LIN {X 0,Y 441.877,Z 678.81,A -85,B 0,C 180,E1 7877.951,E2 7877.951} C_VEL
LIN {X 0,Y 441.94,Z 678.81,A -85,B 0,C 180,E1 7887.839,E2 7887.839} C_VEL
LIN {X 0,Y 441.992,Z 678.81,A -85,B 0,C 180,E1 7896.74,E2 7896.74} C_VEL
LIN {X 0,Y 442.419,Z 678.81,A -85,B 0,C 180,E1 7907.114,E2 7907.114} C_VEL
LIN {X 0,Y 443.093,Z 678.81,A -85,B 0,C 180,E1 7917.053,E2 7917.053} C_VEL
LIN {X 0,Y 442.904,Z 678.81,A -85,B 0,C 180,E1 7928.868,E2 7928.868} C_VEL
LIN {X 0,Y 442.435,Z 678.81,A -85,B 0,C 180,E1 7939.396,E2 7939.396} C_VEL
LIN {X 0,Y 442.136,Z 678.81,A -85,B 0,C 180,E1 7949.846,E2 7949.846} C_VEL
LIN {X 0,Y 441.88,Z 678.81,A -85,B 0,C 180,E1 7959.445,E2 7959.445} C_VEL
LIN {X 0,Y 441.823,Z 678.81,A -85,B 0,C 180,E1 7967.95,E2 7967.95} C_VEL
LIN {X 0,Y 441.903,Z 678.81,A -85,B 0,C 180,E1 7977.84,E2 7977.84} C_VEL
LIN {X 0,Y 441.903,Z 678.81,A -85,B 0,C 180,E1 7986.739,E2 7986.739} C_VEL
LIN {X 0,Y 442.388,Z 678.81,A -85,B 0,C 180,E1 7997.116,E2 7997.116} C_VEL
LIN {X 0,Y 443.106,Z 678.81,A -85,B 0,C 180,E1 8007.055,E2 8007.055} C_VEL
LIN {X 0,Y 442.18,Z 679.143,A -85,B 0,C 180,E1 8012.274,E2 8012.274} C_VEL
LIN {X 0,Y 449.727,Z 716.922,A -85,B 0,C 180,E1 8014.527,E2 8014.527} C_VEL
LIN {X 0,Y 447.081,Z 751.878,A -85,B 0,C 180,E1 8018.049,E2 8018.049} C_VEL
LIN {X 0,Y 445.187,Z 775.919,A -85,B 0,C 180,E1 8022.801,E2 8022.801} C_VEL
LIN {X 0,Y 444.517,Z 785.576,A -85,B 0,C 180,E1 8026.869,E2 8026.869} C_VEL
LIN {X 0,Y 444.32,Z 787.613,A -85,B 0,C 180,E1 8031.016,E2 8031.016} C_VEL
LIN {X 0,Y 445.139,Z 777.632,A -85,B 0,C 180,E1 8036.853,E2 8036.853} C_VEL
LIN {X 0,Y 447.345,Z 753.499,A -85,B 0,C 180,E1 8041.883,E2 8041.883} C_VEL
LIN {X 0,Y 450.088,Z 718.084,A -85,B 0,C 180,E1 8045.554,E2 8045.554} C_VEL
LIN {X 0,Y 445.324,Z 689.075,A -85,B 0,C 180,E1 8047.469,E2 8047.469} C_VEL
LIN {X 0,Y 442.183,Z 678.81,A -85,B 0,C 180,E1 8048.21,E2 8048.21} C_VEL
LIN {X 0,Y 441.838,Z 678.81,A -85,B 0,C 180,E1 8057.952,E2 8057.952} C_VEL
LIN {X 0,Y 441.944,Z 678.81,A -85,B 0,C 180,E1 8067.844,E2 8067.844} C_VEL
LIN {X 0,Y 441.985,Z 678.81,A -85,B 0,C 180,E1 8076.744,E2 8076.744} C_VEL
LIN {X 0,Y 442.41,Z 678.81,A -85,B 0,C 180,E1 8087.118,E2 8087.118} C_VEL
LIN {X 0,Y 443.095,Z 678.81,A -85,B 0,C 180,E1 8097.057,E2 8097.057} C_VEL
LIN {X 0,Y 443.049,Z 678.81,A -85,B 0,C 180,E1 8106.888,E2 8106.888} C_VEL
LIN {X 0,Y 442.491,Z 678.81,A -85,B 0,C 180,E1 8116.952,E2 8116.952} C_VEL
LIN {X 0,Y 442.197,Z 678.81,A -85,B 0,C 180,E1 8127.604,E2 8127.604} C_VEL
LIN {X 0,Y 442.091,Z 678.81,A -85,B 0,C 180,E1 8136.926,E2 8136.926} C_VEL
LIN {X 0,Y 441.903,Z 678.81,A -85,B 0,C 180,E1 8147.596,E2 8147.596} C_VEL
LIN {X 0,Y 441.983,Z 678.81,A -85,B 0,C 180,E1 8157.846,E2 8157.846} C_VEL
LIN {X 0,Y 442.499,Z 680.168,A -85,B 0,C 180,E1 8161.703,E2 8161.703} C_VEL
LIN {X 0,Y 454.771,Z 724.239,A -85,B 0,C 180,E1 8163.121,E2 8163.121} C_VEL
LIN {X 0,Y 452.774,Z 780.472,A -85,B 0,C 180,E1 8164.766,E2 8164.766} C_VEL
LIN {X 0,Y 452.64,Z 781.9,A -85,B 0,C 180,E1 8164.834,E2 8164.834} C_VEL
LIN {X 0,Y 442.739,Z 813.411,A -85,B 0,C 180,E1 8166.492,E2 8166.492} C_VEL
LIN {X 0,Y 438.607,Z 858.556,A -85,B 0,C 180,E1 8171.213,E2 8171.213} C_VEL
LIN {X 0,Y 436.435,Z 891.911,A -85,B 0,C 180,E1 8177.193,E2 8177.193} C_VEL
LIN {X 0,Y 436.07,Z 912.085,A -85,B 0,C 180,E1 8184.007,E2 8184.007} C_VEL
LIN {X 0,Y 435.871,Z 917.371,A -85,B 0,C 180,E1 8190.997,E2 8190.997} C_VEL
LIN {X 0,Y 435.685,Z 909.052,A -85,B 0,C 180,E1 8197.505,E2 8197.505} C_VEL
LIN {X 0,Y 436.677,Z 886.527,A -85,B 0,C 180,E1 8204.079,E2 8204.079} C_VEL
LIN {X 0,Y 439.545,Z 849.957,A -85,B 0,C 180,E1 8209.934,E2 8209.934} C_VEL
LIN {X 0,Y 443.584,Z 803.083,A -85,B 0,C 180,E1 8214.238,E2 8214.238} C_VEL
LIN {X 0,Y 446.827,Z 750.347,A -85,B 0,C 180,E1 8216.674,E2 8216.674} C_VEL
LIN {X 0,Y 444.835,Z 713.614,A -85,B 0,C 180,E1 8217.491,E2 8217.491} C_VEL
LIN {X 0,Y 433.969,Z 678.81,A -85,B 0,C 180,E1 8218.814,E2 8218.814} C_VEL
LIN {X 0,Y 433.799,Z 678.81,A -85,B 0,C 180,E1 8228.076,E2 8228.076} C_VEL
LIN {X 0,Y 433.797,Z 678.81,A -85,B 0,C 180,E1 8238.775,E2 8238.775} C_VEL
LIN {X 0,Y 433.951,Z 678.81,A -85,B 0,C 180,E1 8249.527,E2 8249.527} C_VEL
LIN {X 0,Y 434.098,Z 678.81,A -85,B 0,C 180,E1 8260.6,E2 8260.6} C_VEL
LIN {X 0,Y 434.846,Z 678.81,A -85,B 0,C 180,E1 8270.962,E2 8270.962} C_VEL
LIN {X 0,Y 435.297,Z 678.81,A -85,B 0,C 180,E1 8278.999,E2 8278.999} C_VEL
LIN {X 0,Y 434.769,Z 678.81,A -85,B 0,C 180,E1 8291.067,E2 8291.067} C_VEL
LIN {X 0,Y 434.349,Z 678.81,A -85,B 0,C 180,E1 8301.521,E2 8301.521} C_VEL
LIN {X 0,Y 433.969,Z 678.81,A -85,B 0,C 180,E1 8311.048,E2 8311.048} C_VEL
LIN {X 0,Y 433.777,Z 678.81,A -85,B 0,C 180,E1 8321.222,E2 8321.222} C_VEL
LIN {X 0,Y 433.68,Z 678.81,A -85,B 0,C 180,E1 8331.937,E2 8331.937} C_VEL
LIN {X 0,Y 433.976,Z 678.81,A -85,B 0,C 180,E1 8341.831,E2 8341.831} C_VEL
LIN {X 0,Y 434.276,Z 678.81,A -85,B 0,C 180,E1 8352.721,E2 8352.721} C_VEL
LIN {X 0,Y 434.938,Z 678.81,A -85,B 0,C 180,E1 8362.986,E2 8362.986} C_VEL
LIN {X 0,Y 434.25,Z 678.81,A -85,B 0,C 180,E1 8371.815,E2 8371.815} C_VEL
LIN {X 0,Y 442.066,Z 718.948,A -85,B 0,C 180,E1 8374.298,E2 8374.298} C_VEL
LIN {X 0,Y 439.279,Z 753.815,A -85,B 0,C 180,E1 8377.943,E2 8377.943} C_VEL
LIN {X 0,Y 437.249,Z 778.246,A -85,B 0,C 180,E1 8383.038,E2 8383.038} C_VEL
LIN {X 0,Y 436.541,Z 787.188,A -85,B 0,C 180,E1 8387.187,E2 8387.187} C_VEL
LIN {X 0,Y 436.779,Z 786.5,A -85,B 0,C 180,E1 8393.551,E2 8393.551} C_VEL
LIN {X 0,Y 438.438,Z 770.38,A -85,B 0,C 180,E1 8399.269,E2 8399.269} C_VEL
LIN {X 0,Y 441.15,Z 741.521,A -85,B 0,C 180,E1 8403.838,E2 8403.838} C_VEL
LIN {X 0,Y 441.511,Z 704.131,A -85,B 0,C 180,E1 8406.978,E2 8406.978} C_VEL
LIN {X 0,Y 434.104,Z 678.81,A -85,B 0,C 180,E1 8408.703,E2 8408.703} C_VEL
LIN {X 0,Y 433.703,Z 678.81,A -85,B 0,C 180,E1 8419.66,E2 8419.66} C_VEL
LIN {X 0,Y 433.978,Z 678.81,A -85,B 0,C 180,E1 8429.534,E2 8429.534} C_VEL
LIN {X 0,Y 434.092,Z 678.81,A -85,B 0,C 180,E1 8440.604,E2 8440.604} C_VEL
LIN {X 0,Y 434.849,Z 678.81,A -85,B 0,C 180,E1 8450.966,E2 8450.966} C_VEL
LIN {X 0,Y 435.015,Z 678.81,A -85,B 0,C 180,E1 8461.002,E2 8461.002} C_VEL
LIN {X 0,Y 434.693,Z 678.81,A -85,B 0,C 180,E1 8471.073,E2 8471.073} C_VEL
LIN {X 0,Y 434.356,Z 678.81,A -85,B 0,C 180,E1 8481.525,E2 8481.525} C_VEL
LIN {X 0,Y 434.026,Z 678.81,A -85,B 0,C 180,E1 8491.06,E2 8491.06} C_VEL
LIN {X 0,Y 433.912,Z 678.81,A -85,B 0,C 180,E1 8501.242,E2 8501.242} C_VEL
LIN {X 0,Y 433.872,Z 678.81,A -85,B 0,C 180,E1 8512.259,E2 8512.259} C_VEL
LIN {X 0,Y 434.464,Z 680.417,A -85,B 0,C 180,E1 8521.215,E2 8521.215} C_VEL
LIN {X 0,Y 447.42,Z 725.661,A -85,B 0,C 180,E1 8522.749,E2 8522.749} C_VEL
LIN {X 0,Y 445.189,Z 781.406,A -85,B 0,C 180,E1 8524.463,E2 8524.463} C_VEL
LIN {X 0,Y 442.739,Z 813.411,A -85,B 0,C 180,E1 8526.492,E2 8526.492} C_VEL
LIN {X 0,Y 432.436,Z 841.873,A -85,B 0,C 180,E1 8528.923,E2 8528.923} C_VEL
LIN {X 0,Y 429.299,Z 879.992,A -85,B 0,C 180,E1 8534.626,E2 8534.626} C_VEL
LIN {X 0,Y 427.929,Z 905.255,A -85,B 0,C 180,E1 8541.332,E2 8541.332} C_VEL
LIN {X 0,Y 427.867,Z 914.935,A -85,B 0,C 180,E1 8546.95,E2 8546.95} C_VEL
LIN {X 0,Y 428.123,Z 913.998,A -85,B 0,C 180,E1 8554.065,E2 8554.065} C_VEL
LIN {X 0,Y 428.103,Z 897.643,A -85,B 0,C 180,E1 8561.243,E2 8561.243} C_VEL
LIN {X 0,Y 429.981,Z 868.516,A -85,B 0,C 180,E1 8567.457,E2 8567.457} C_VEL
LIN {X 0,Y 433.947,Z 825.892,A -85,B 0,C 180,E1 8572.695,E2 8572.695} C_VEL
LIN {X 0,Y 438.014,Z 774.746,A -85,B 0,C 180,E1 8576.137,E2 8576.137} C_VEL
LIN {X 0,Y 438.357,Z 718.264,A -85,B 0,C 180,E1 8577.745,E2 8577.745} C_VEL
LIN {X 0,Y 425.957,Z 678.81,A -85,B 0,C 180,E1 8579.198,E2 8579.198} C_VEL
LIN {X 0,Y 425.769,Z 678.81,A -85,B 0,C 180,E1 8589.969,E2 8589.969} C_VEL
LIN {X 0,Y 425.735,Z 678.81,A -85,B 0,C 180,E1 8600.029,E2 8600.029} C_VEL
LIN {X 0,Y 425.916,Z 678.81,A -85,B 0,C 180,E1 8610.802,E2 8610.802} C_VEL
LIN {X 0,Y 426.102,Z 678.81,A -85,B 0,C 180,E1 8620.697,E2 8620.697} C_VEL
LIN {X 0,Y 426.796,Z 678.81,A -85,B 0,C 180,E1 8630.79,E2 8630.79} C_VEL
LIN {X 0,Y 427.307,Z 678.81,A -85,B 0,C 180,E1 8638.98,E2 8638.98} C_VEL
LIN {X 0,Y 426.731,Z 678.81,A -85,B 0,C 180,E1 8651.278,E2 8651.278} C_VEL
LIN {X 0,Y 426.325,Z 678.81,A -85,B 0,C 180,E1 8661.947,E2 8661.947} C_VEL
LIN {X 0,Y 425.888,Z 678.81,A -85,B 0,C 180,E1 8673.137,E2 8673.137} C_VEL
LIN {X 0,Y 425.745,Z 678.81,A -85,B 0,C 180,E1 8684.033,E2 8684.033} C_VEL
LIN {X 0,Y 425.692,Z 678.81,A -85,B 0,C 180,E1 8693.97,E2 8693.97} C_VEL
LIN {X 0,Y 425.958,Z 678.81,A -85,B 0,C 180,E1 8703.555,E2 8703.555} C_VEL
LIN {X 0,Y 426.356,Z 678.81,A -85,B 0,C 180,E1 8714.517,E2 8714.517} C_VEL
LIN {X 0,Y 426.839,Z 678.81,A -85,B 0,C 180,E1 8724.901,E2 8724.901} C_VEL
LIN {X 0,Y 426.588,Z 680.772,A -85,B 0,C 180,E1 8731.51,E2 8731.51} C_VEL
LIN {X 0,Y 434.61,Z 718.951,A -85,B 0,C 180,E1 8733.914,E2 8733.914} C_VEL
LIN {X 0,Y 431.635,Z 753.982,A -85,B 0,C 180,E1 8737.576,E2 8737.576} C_VEL
LIN {X 0,Y 429.438,Z 778.919,A -85,B 0,C 180,E1 8742.76,E2 8742.76} C_VEL
LIN {X 0,Y 428.589,Z 788.786,A -85,B 0,C 180,E1 8747.516,E2 8747.516} C_VEL
LIN {X 0,Y 428.848,Z 788.247,A -85,B 0,C 180,E1 8753.23,E2 8753.23} C_VEL
LIN {X 0,Y 430.38,Z 773.875,A -85,B 0,C 180,E1 8758.929,E2 8758.929} C_VEL
LIN {X 0,Y 433.163,Z 747.105,A -85,B 0,C 180,E1 8763.627,E2 8763.627} C_VEL
LIN {X 0,Y 435.057,Z 709.963,A -85,B 0,C 180,E1 8767.024,E2 8767.024} C_VEL
LIN {X 0,Y 426.081,Z 678.81,A -85,B 0,C 180,E1 8769.062,E2 8769.062} C_VEL
LIN {X 0,Y 425.673,Z 678.81,A -85,B 0,C 180,E1 8780.039,E2 8780.039} C_VEL
LIN {X 0,Y 425.971,Z 678.81,A -85,B 0,C 180,E1 8791.253,E2 8791.253} C_VEL
LIN {X 0,Y 426.21,Z 678.81,A -85,B 0,C 180,E1 8802.384,E2 8802.384} C_VEL
LIN {X 0,Y 426.906,Z 678.81,A -85,B 0,C 180,E1 8812.855,E2 8812.855} C_VEL
LIN {X 0,Y 427.024,Z 678.81,A -85,B 0,C 180,E1 8821.02,E2 8821.02} C_VEL
LIN {X 0,Y 426.672,Z 678.81,A -85,B 0,C 180,E1 8831.284,E2 8831.284} C_VEL
LIN {X 0,Y 426.324,Z 678.81,A -85,B 0,C 180,E1 8841.951,E2 8841.951} C_VEL
LIN {X 0,Y 426.006,Z 678.81,A -85,B 0,C 180,E1 8853.161,E2 8853.161} C_VEL
LIN {X 0,Y 425.864,Z 678.81,A -85,B 0,C 180,E1 8864.023,E2 8864.023} C_VEL
LIN {X 0,Y 425.827,Z 678.81,A -85,B 0,C 180,E1 8873.983,E2 8873.983} C_VEL
LIN {X 0,Y 426.385,Z 680.424,A -85,B 0,C 180,E1 8880.699,E2 8880.699} C_VEL
LIN {X 0,Y 440.084,Z 727.574,A -85,B 0,C 180,E1 8882.364,E2 8882.364} C_VEL
LIN {X 0,Y 437.615,Z 782.033,A -85,B 0,C 180,E1 8884.133,E2 8884.133} C_VEL
LIN {X 0,Y 433.379,Z 832.186,A -85,B 0,C 180,E1 8887.881,E2 8887.881} C_VEL
LIN {X 0,Y 432.436,Z 841.873,A -85,B 0,C 180,E1 8888.923,E2 8888.923} C_VEL
LIN {X 0,Y 422.308,Z 866.311,A -85,B 0,C 180,E1 8892.084,E2 8892.084} C_VEL
LIN {X 0,Y 420.41,Z 896.275,A -85,B 0,C 180,E1 8898.549,E2 8898.549} C_VEL
LIN {X 0,Y 420.05,Z 912.726,A -85,B 0,C 180,E1 8905.856,E2 8905.856} C_VEL
LIN {X 0,Y 420.028,Z 915.036,A -85,B 0,C 180,E1 8911.035,E2 8911.035} C_VEL
LIN {X 0,Y 419.87,Z 906.627,A -85,B 0,C 180,E1 8917.79,E2 8917.79} C_VEL
LIN {X 0,Y 421.133,Z 882.605,A -85,B 0,C 180,E1 8924.877,E2 8924.877} C_VEL
LIN {X 0,Y 424.28,Z 845.522,A -85,B 0,C 180,E1 8930.82,E2 8930.82} C_VEL
LIN {X 0,Y 428.604,Z 798.386,A -85,B 0,C 180,E1 8935.148,E2 8935.148} C_VEL
LIN {X 0,Y 432.027,Z 745.581,A -85,B 0,C 180,E1 8937.527,E2 8937.527} C_VEL
LIN {X 0,Y 429.827,Z 716.725,A -85,B 0,C 180,E1 8938.211,E2 8938.211} C_VEL
LIN {X 0,Y 417.896,Z 678.81,A -85,B 0,C 180,E1 8939.608,E2 8939.608} C_VEL
LIN {X 0,Y 417.75,Z 678.81,A -85,B 0,C 180,E1 8949.473,E2 8949.473} C_VEL
LIN {X 0,Y 417.709,Z 678.81,A -85,B 0,C 180,E1 8960.517,E2 8960.517} C_VEL
LIN {X 0,Y 417.92,Z 678.81,A -85,B 0,C 180,E1 8970.641,E2 8970.641} C_VEL
LIN {X 0,Y 418.163,Z 678.81,A -85,B 0,C 180,E1 8982.03,E2 8982.03} C_VEL
LIN {X 0,Y 418.885,Z 678.81,A -85,B 0,C 180,E1 8992.713,E2 8992.713} C_VEL
LIN {X 0,Y 418.382,Z 678.81,A -85,B 0,C 180,E1 9001.037,E2 9001.037} C_VEL
LIN {X 0,Y 418.714,Z 678.81,A -85,B 0,C 180,E1 9011.497,E2 9011.497} C_VEL
LIN {X 0,Y 418.276,Z 678.81,A -85,B 0,C 180,E1 9022.392,E2 9022.392} C_VEL
LIN {X 0,Y 417.879,Z 678.81,A -85,B 0,C 180,E1 9031.774,E2 9031.774} C_VEL
LIN {X 0,Y 417.759,Z 678.81,A -85,B 0,C 180,E1 9042.224,E2 9042.224} C_VEL
LIN {X 0,Y 417.634,Z 678.81,A -85,B 0,C 180,E1 9053.162,E2 9053.162} C_VEL
LIN {X 0,Y 417.879,Z 678.81,A -85,B 0,C 180,E1 9063.003,E2 9063.003} C_VEL
LIN {X 0,Y 418.297,Z 678.81,A -85,B 0,C 180,E1 9074.211,E2 9074.211} C_VEL
LIN {X 0,Y 418.87,Z 678.81,A -85,B 0,C 180,E1 9085.09,E2 9085.09} C_VEL
LIN {X 0,Y 418.64,Z 680.586,A -85,B 0,C 180,E1 9091.071,E2 9091.071} C_VEL
LIN {X 0,Y 426.982,Z 720.646,A -85,B 0,C 180,E1 9093.651,E2 9093.651} C_VEL
LIN {X 0,Y 423.848,Z 755.871,A -85,B 0,C 180,E1 9097.458,E2 9097.458} C_VEL
LIN {X 0,Y 421.626,Z 779.548,A -85,B 0,C 180,E1 9102.472,E2 9102.472} C_VEL
LIN {X 0,Y 420.642,Z 790.276,A -85,B 0,C 180,E1 9107.858,E2 9107.858} C_VEL
LIN {X 0,Y 421.163,Z 787.758,A -85,B 0,C 180,E1 9114.48,E2 9114.48} C_VEL
LIN {X 0,Y 423.17,Z 770.87,A -85,B 0,C 180,E1 9120.146,E2 9120.146} C_VEL
LIN {X 0,Y 426.466,Z 740.702,A -85,B 0,C 180,E1 9124.85,E2 9124.85} C_VEL
LIN {X 0,Y 426.787,Z 707.886,A -85,B 0,C 180,E1 9127.692,E2 9127.692} C_VEL
LIN {X 0,Y 417.978,Z 678.81,A -85,B 0,C 180,E1 9129.784,E2 9129.784} C_VEL
LIN {X 0,Y 417.648,Z 678.81,A -85,B 0,C 180,E1 9140.515,E2 9140.515} C_VEL
LIN {X 0,Y 417.94,Z 678.81,A -85,B 0,C 180,E1 9150.648,E2 9150.648} C_VEL
LIN {X 0,Y 418.157,Z 678.81,A -85,B 0,C 180,E1 9162.034,E2 9162.034} C_VEL
LIN {X 0,Y 418.883,Z 678.81,A -85,B 0,C 180,E1 9172.717,E2 9172.717} C_VEL
LIN {X 0,Y 419.018,Z 678.81,A -85,B 0,C 180,E1 9181.04,E2 9181.04} C_VEL
LIN {X 0,Y 418.673,Z 678.81,A -85,B 0,C 180,E1 9191.502,E2 9191.502} C_VEL
LIN {X 0,Y 418.25,Z 678.81,A -85,B 0,C 180,E1 9202.398,E2 9202.398} C_VEL
LIN {X 0,Y 417.956,Z 678.81,A -85,B 0,C 180,E1 9211.772,E2 9211.772} C_VEL
LIN {X 0,Y 417.866,Z 678.81,A -85,B 0,C 180,E1 9222.216,E2 9222.216} C_VEL
LIN {X 0,Y 417.827,Z 678.81,A -85,B 0,C 180,E1 9233.182,E2 9233.182} C_VEL
LIN {X 0,Y 418.227,Z 680.028,A -85,B 0,C 180,E1 9240.136,E2 9240.136} C_VEL
LIN {X 0,Y 432.824,Z 725.086,A -85,B 0,C 180,E1 9241.887,E2 9241.887} C_VEL
LIN {X 0,Y 430.313,Z 780.291,A -85,B 0,C 180,E1 9243.661,E2 9243.661} C_VEL
LIN {X 0,Y 425.889,Z 829.452,A -85,B 0,C 180,E1 9247.339,E2 9247.339} C_VEL
LIN {X 0,Y 422.308,Z 866.311,A -85,B 0,C 180,E1 9252.084,E2 9252.084} C_VEL
LIN {X 0,Y 412.639,Z 886.088,A -85,B 0,C 180,E1 9255.928,E2 9255.928} C_VEL
LIN {X 0,Y 412.034,Z 906.463,A -85,B 0,C 180,E1 9262.593,E2 9262.593} C_VEL
LIN {X 0,Y 412.474,Z 913.896,A -85,B 0,C 180,E1 9268.946,E2 9268.946} C_VEL
LIN {X 0,Y 411.927,Z 908.513,A -85,B 0,C 180,E1 9276.37,E2 9276.37} C_VEL
LIN {X 0,Y 412.395,Z 889.677,A -85,B 0,C 180,E1 9283.164,E2 9283.164} C_VEL
LIN {X 0,Y 415.027,Z 856.773,A -85,B 0,C 180,E1 9289.491,E2 9289.491} C_VEL
LIN {X 0,Y 419.621,Z 812.108,A -85,B 0,C 180,E1 9294.433,E2 9294.433} C_VEL
LIN {X 0,Y 423.803,Z 760.344,A -85,B 0,C 180,E1 9297.434,E2 9297.434} C_VEL
LIN {X 0,Y 422.852,Z 719.81,A -85,B 0,C 180,E1 9298.527,E2 9298.527} C_VEL
LIN {X 0,Y 409.873,Z 678.81,A -85,B 0,C 180,E1 9299.989,E2 9299.989} C_VEL
LIN {X 0,Y 409.683,Z 678.81,A -85,B 0,C 180,E1 9310.585,E2 9310.585} C_VEL
LIN {X 0,Y 409.657,Z 678.81,A -85,B 0,C 180,E1 9319.583,E2 9319.583} C_VEL
LIN {X 0,Y 409.898,Z 678.81,A -85,B 0,C 180,E1 9330.462,E2 9330.462} C_VEL
LIN {X 0,Y 410.087,Z 678.81,A -85,B 0,C 180,E1 9341.663,E2 9341.663} C_VEL
LIN {X 0,Y 410.856,Z 678.81,A -85,B 0,C 180,E1 9352.57,E2 9352.57} C_VEL
LIN {X 0,Y 410.387,Z 678.81,A -85,B 0,C 180,E1 9361.057,E2 9361.057} C_VEL
LIN {X 0,Y 410.68,Z 678.81,A -85,B 0,C 180,E1 9371.725,E2 9371.725} C_VEL
LIN {X 0,Y 410.214,Z 678.81,A -85,B 0,C 180,E1 9382.856,E2 9382.856} C_VEL
LIN {X 0,Y 409.699,Z 678.81,A -85,B 0,C 180,E1 9393.549,E2 9393.549} C_VEL
LIN {X 0,Y 409.614,Z 678.81,A -85,B 0,C 180,E1 9403.744,E2 9403.744} C_VEL
LIN {X 0,Y 409.647,Z 678.81,A -85,B 0,C 180,E1 9414.956,E2 9414.956} C_VEL
LIN {X 0,Y 409.871,Z 678.81,A -85,B 0,C 180,E1 9425.111,E2 9425.111} C_VEL
LIN {X 0,Y 410.281,Z 678.81,A -85,B 0,C 180,E1 9436.089,E2 9436.089} C_VEL
LIN {X 0,Y 411.052,Z 678.81,A -85,B 0,C 180,E1 9446.826,E2 9446.826} C_VEL
LIN {X 0,Y 410.8,Z 680.679,A -85,B 0,C 180,E1 9450.628,E2 9450.628} C_VEL
LIN {X 0,Y 419.439,Z 721.598,A -85,B 0,C 180,E1 9453.324,E2 9453.324} C_VEL
LIN {X 0,Y 416.055,Z 757.722,A -85,B 0,C 180,E1 9457.335,E2 9457.335} C_VEL
LIN {X 0,Y 413.722,Z 781.326,A -85,B 0,C 180,E1 9462.551,E2 9462.551} C_VEL
LIN {X 0,Y 412.702,Z 791.758,A -85,B 0,C 180,E1 9468.213,E2 9468.213} C_VEL
LIN {X 0,Y 413.373,Z 788.324,A -85,B 0,C 180,E1 9474.972,E2 9474.972} C_VEL
LIN {X 0,Y 415.696,Z 769.725,A -85,B 0,C 180,E1 9480.918,E2 9480.918} C_VEL
LIN {X 0,Y 419.251,Z 739.415,A -85,B 0,C 180,E1 9485.469,E2 9485.469} C_VEL
LIN {X 0,Y 419.264,Z 708.889,A -85,B 0,C 180,E1 9488.14,E2 9488.14} C_VEL
LIN {X 0,Y 409.899,Z 678.81,A -85,B 0,C 180,E1 9490.383,E2 9490.383} C_VEL
LIN {X 0,Y 409.607,Z 678.81,A -85,B 0,C 180,E1 9499.582,E2 9499.582} C_VEL
LIN {X 0,Y 409.928,Z 678.81,A -85,B 0,C 180,E1 9510.455,E2 9510.455} C_VEL
LIN {X 0,Y 410.08,Z 678.81,A -85,B 0,C 180,E1 9521.667,E2 9521.667} C_VEL
LIN {X 0,Y 410.855,Z 678.81,A -85,B 0,C 180,E1 9532.574,E2 9532.574} C_VEL
LIN {X 0,Y 411.028,Z 678.81,A -85,B 0,C 180,E1 9541.06,E2 9541.06} C_VEL
LIN {X 0,Y 410.659,Z 678.81,A -85,B 0,C 180,E1 9551.73,E2 9551.73} C_VEL
LIN {X 0,Y 410.186,Z 678.81,A -85,B 0,C 180,E1 9562.863,E2 9562.863} C_VEL
LIN {X 0,Y 409.857,Z 678.81,A -85,B 0,C 180,E1 9573.582,E2 9573.582} C_VEL
LIN {X 0,Y 409.724,Z 678.81,A -85,B 0,C 180,E1 9583.76,E2 9583.76} C_VEL
LIN {X 0,Y 409.762,Z 678.81,A -85,B 0,C 180,E1 9594.967,E2 9594.967} C_VEL
LIN {X 0,Y 410.166,Z 679.993,A -85,B 0,C 180,E1 9599.556,E2 9599.556} C_VEL
LIN {X 0,Y 425.551,Z 729.625,A -85,B 0,C 180,E1 9601.516,E2 9601.516} C_VEL
LIN {X 0,Y 422.517,Z 784.176,A -85,B 0,C 180,E1 9603.472,E2 9603.472} C_VEL
LIN {X 0,Y 417.781,Z 833.169,A -85,B 0,C 180,E1 9607.439,E2 9607.439} C_VEL
LIN {X 0,Y 413.943,Z 873.737,A -85,B 0,C 180,E1 9613.297,E2 9613.297} C_VEL
LIN {X 0,Y 412.639,Z 886.088,A -85,B 0,C 180,E1 9615.928,E2 9615.928} C_VEL
LIN {X 0,Y 404.245,Z 900.452,A -85,B 0,C 180,E1 9620.347,E2 9620.347} C_VEL
LIN {X 0,Y 404.134,Z 911.436,A -85,B 0,C 180,E1 9626.771,E2 9626.771} C_VEL
LIN {X 0,Y 404.199,Z 911.459,A -85,B 0,C 180,E1 9633.228,E2 9633.228} C_VEL
LIN {X 0,Y 404.31,Z 898.79,A -85,B 0,C 180,E1 9640.27,E2 9640.27} C_VEL
LIN {X 0,Y 405.941,Z 870.844,A -85,B 0,C 180,E1 9647.283,E2 9647.283} C_VEL
LIN {X 0,Y 410.172,Z 830.21,A -85,B 0,C 180,E1 9653.004,E2 9653.004} C_VEL
LIN {X 0,Y 414.832,Z 780.362,A -85,B 0,C 180,E1 9656.893,E2 9656.893} C_VEL
LIN {X 0,Y 416.687,Z 725.301,A -85,B 0,C 180,E1 9658.767,E2 9658.767} C_VEL
LIN {X 0,Y 401.757,Z 678.81,A -85,B 0,C 180,E1 9660.659,E2 9660.659} C_VEL
LIN {X 0,Y 401.59,Z 678.81,A -85,B 0,C 180,E1 9671.399,E2 9671.399} C_VEL
LIN {X 0,Y 401.559,Z 678.81,A -85,B 0,C 180,E1 9681.418,E2 9681.418} C_VEL
LIN {X 0,Y 401.914,Z 678.81,A -85,B 0,C 180,E1 9692.537,E2 9692.537} C_VEL
LIN {X 0,Y 402.243,Z 678.81,A -85,B 0,C 180,E1 9704.162,E2 9704.162} C_VEL
LIN {X 0,Y 402.811,Z 678.81,A -85,B 0,C 180,E1 9714.593,E2 9714.593} C_VEL
LIN {X 0,Y 402.082,Z 678.81,A -85,B 0,C 180,E1 9723.243,E2 9723.243} C_VEL
LIN {X 0,Y 402.638,Z 678.81,A -85,B 0,C 180,E1 9731.962,E2 9731.962} C_VEL
LIN {X 0,Y 402.187,Z 678.81,A -85,B 0,C 180,E1 9743.339,E2 9743.339} C_VEL
LIN {X 0,Y 401.715,Z 678.81,A -85,B 0,C 180,E1 9753.213,E2 9753.213} C_VEL
LIN {X 0,Y 401.548,Z 678.81,A -85,B 0,C 180,E1 9764.36,E2 9764.36} C_VEL
LIN {X 0,Y 401.597,Z 678.81,A -85,B 0,C 180,E1 9774.335,E2 9774.335} C_VEL
LIN {X 0,Y 401.801,Z 678.81,A -85,B 0,C 180,E1 9784.257,E2 9784.257} C_VEL
LIN {X 0,Y 402.245,Z 678.81,A -85,B 0,C 180,E1 9795.805,E2 9795.805} C_VEL
LIN {X 0,Y 403.055,Z 678.81,A -85,B 0,C 180,E1 9806.762,E2 9806.762} C_VEL
LIN {X 0,Y 402.835,Z 679.598,A -85,B 0,C 180,E1 9810.135,E2 9810.135} C_VEL
LIN {X 0,Y 412.006,Z 721.097,A -85,B 0,C 180,E1 9812.871,E2 9812.871} C_VEL
LIN {X 0,Y 408.434,Z 757.824,A -85,B 0,C 180,E1 9816.936,E2 9816.936} C_VEL
LIN {X 0,Y 405.919,Z 782.043,A -85,B 0,C 180,E1 9822.278,E2 9822.278} C_VEL
LIN {X 0,Y 404.783,Z 793.151,A -85,B 0,C 180,E1 9828.582,E2 9828.582} C_VEL
LIN {X 0,Y 405.57,Z 788.863,A -85,B 0,C 180,E1 9835.487,E2 9835.487} C_VEL
LIN {X 0,Y 408.128,Z 769.979,A -85,B 0,C 180,E1 9841.387,E2 9841.387} C_VEL
LIN {X 0,Y 411.972,Z 739.194,A -85,B 0,C 180,E1 9845.998,E2 9845.998} C_VEL
LIN {X 0,Y 411.687,Z 709.442,A -85,B 0,C 180,E1 9848.647,E2 9848.647} C_VEL
LIN {X 0,Y 401.821,Z 678.81,A -85,B 0,C 180,E1 9850.932,E2 9850.932} C_VEL
LIN {X 0,Y 401.501,Z 678.81,A -85,B 0,C 180,E1 9861.417,E2 9861.417} C_VEL
LIN {X 0,Y 401.922,Z 678.81,A -85,B 0,C 180,E1 9872.535,E2 9872.535} C_VEL
LIN {X 0,Y 402.241,Z 678.81,A -85,B 0,C 180,E1 9884.164,E2 9884.164} C_VEL
LIN {X 0,Y 402.812,Z 678.81,A -85,B 0,C 180,E1 9894.598,E2 9894.598} C_VEL
LIN {X 0,Y 402.885,Z 678.81,A -85,B 0,C 180,E1 9903.46,E2 9903.46} C_VEL
LIN {X 0,Y 402.541,Z 678.81,A -85,B 0,C 180,E1 9914.188,E2 9914.188} C_VEL
LIN {X 0,Y 402.045,Z 678.81,A -85,B 0,C 180,E1 9925.73,E2 9925.73} C_VEL
LIN {X 0,Y 401.867,Z 678.81,A -85,B 0,C 180,E1 9935.83,E2 9935.83} C_VEL
LIN {X 0,Y 401.635,Z 678.81,A -85,B 0,C 180,E1 9947.466,E2 9947.466} C_VEL
LIN {X 0,Y 402.087,Z 679.93,A -85,B 0,C 180,E1 9958.948,E2 9958.948} C_VEL
LIN {X 0,Y 418.318,Z 730.642,A -85,B 0,C 180,E1 9961.07,E2 9961.07} C_VEL
LIN {X 0,Y 415.075,Z 784.371,A -85,B 0,C 180,E1 9963.079,E2 9963.079} C_VEL
LIN {X 0,Y 410.064,Z 833.053,A -85,B 0,C 180,E1 9967.134,E2 9967.134} C_VEL
LIN {X 0,Y 406.053,Z 872.679,A -85,B 0,C 180,E1 9973.002,E2 9973.002} C_VEL
LIN {X 0,Y 404.261,Z 900.262,A -85,B 0,C 180,E1 9980.275,E2 9980.275} C_VEL
LIN {X 0,Y 404.245,Z 900.452,A -85,B 0,C 180,E1 9980.347,E2 9980.347} C_VEL
LIN {X 0,Y 396.315,Z 908.704,A -85,B 0,C 180,E1 9985.174,E2 9985.174} C_VEL
LIN {X 0,Y 396.284,Z 911.524,A -85,B 0,C 180,E1 9991.097,E2 9991.097} C_VEL
LIN {X 0,Y 396.117,Z 902.885,A -85,B 0,C 180,E1 9998.26,E2 9998.26} C_VEL
LIN {X 0,Y 397.622,Z 878.358,A -85,B 0,C 180,E1 10005.779,E2 10005.779} C_VEL
LIN {X 0,Y 401.185,Z 841.339,A -85,B 0,C 180,E1 10011.935,E2 10011.935} C_VEL
LIN {X 0,Y 406.117,Z 793.562,A -85,B 0,C 180,E1 10016.44,E2 10016.44} C_VEL
LIN {X 0,Y 409.771,Z 741.027,A -85,B 0,C 180,E1 10018.812,E2 10018.812} C_VEL
LIN {X 0,Y 406.222,Z 717.194,A -85,B 0,C 180,E1 10019.503,E2 10019.503} C_VEL
LIN {X 0,Y 393.732,Z 678.81,A -85,B 0,C 180,E1 10021.162,E2 10021.162} C_VEL
LIN {X 0,Y 393.584,Z 678.81,A -85,B 0,C 180,E1 10032.435,E2 10032.435} C_VEL
LIN {X 0,Y 393.515,Z 678.81,A -85,B 0,C 180,E1 10043.287,E2 10043.287} C_VEL
LIN {X 0,Y 393.861,Z 678.81,A -85,B 0,C 180,E1 10053.694,E2 10053.694} C_VEL
LIN {X 0,Y 394.249,Z 678.81,A -85,B 0,C 180,E1 10065.508,E2 10065.508} C_VEL
LIN {X 0,Y 395.03,Z 678.81,A -85,B 0,C 180,E1 10076.694,E2 10076.694} C_VEL
LIN {X 0,Y 394.728,Z 678.81,A -85,B 0,C 180,E1 10089.961,E2 10089.961} C_VEL
LIN {X 0,Y 394.222,Z 678.81,A -85,B 0,C 180,E1 10101.45,E2 10101.45} C_VEL
LIN {X 0,Y 393.755,Z 678.81,A -85,B 0,C 180,E1 10111.351,E2 10111.351} C_VEL
LIN {X 0,Y 393.549,Z 678.81,A -85,B 0,C 180,E1 10122.439,E2 10122.439} C_VEL
LIN {X 0,Y 393.464,Z 678.81,A -85,B 0,C 180,E1 10133.286,E2 10133.286} C_VEL
LIN {X 0,Y 393.804,Z 678.81,A -85,B 0,C 180,E1 10143.695,E2 10143.695} C_VEL
LIN {X 0,Y 394.234,Z 678.81,A -85,B 0,C 180,E1 10155.51,E2 10155.51} C_VEL
LIN {X 0,Y 395.053,Z 678.81,A -85,B 0,C 180,E1 10166.697,E2 10166.697} C_VEL
LIN {X 0,Y 394.973,Z 679.345,A -85,B 0,C 180,E1 10169.656,E2 10169.656} C_VEL
LIN {X 0,Y 404.392,Z 723.106,A -85,B 0,C 180,E1 10172.603,E2 10172.603} C_VEL
LIN {X 0,Y 400.658,Z 759.671,A -85,B 0,C 180,E1 10176.798,E2 10176.798} C_VEL
LIN {X 0,Y 398.099,Z 783.063,A -85,B 0,C 180,E1 10182.102,E2 10182.102} C_VEL
LIN {X 0,Y 397.132,Z 792.557,A -85,B 0,C 180,E1 10186.654,E2 10186.654} C_VEL
LIN {X 0,Y 396.917,Z 794.672,A -85,B 0,C 180,E1 10191.298,E2 10191.298} C_VEL
LIN {X 0,Y 398.34,Z 785.062,A -85,B 0,C 180,E1 10197.854,E2 10197.854} C_VEL
LIN {X 0,Y 401.691,Z 761.881,A -85,B 0,C 180,E1 10203.473,E2 10203.473} C_VEL
LIN {X 0,Y 405.902,Z 725.808,A -85,B 0,C 180,E1 10207.807,E2 10207.807} C_VEL
LIN {X 0,Y 397.775,Z 690.073,A -85,B 0,C 180,E1 10210.734,E2 10210.734} C_VEL
LIN {X 0,Y 393.727,Z 678.81,A -85,B 0,C 180,E1 10211.585,E2 10211.585} C_VEL
LIN {X 0,Y 393.435,Z 678.81,A -85,B 0,C 180,E1 10222.253,E2 10222.253} C_VEL
LIN {X 0,Y 393.864,Z 678.81,A -85,B 0,C 180,E1 10233.7,E2 10233.7} C_VEL
LIN {X 0,Y 394.24,Z 678.81,A -85,B 0,C 180,E1 10245.512,E2 10245.512} C_VEL
LIN {X 0,Y 395.029,Z 678.81,A -85,B 0,C 180,E1 10256.699,E2 10256.699} C_VEL
LIN {X 0,Y 394.887,Z 678.81,A -85,B 0,C 180,E1 10267.733,E2 10267.733} C_VEL
LIN {X 0,Y 394.257,Z 678.81,A -85,B 0,C 180,E1 10279.101,E2 10279.101} C_VEL
LIN {X 0,Y 393.841,Z 678.81,A -85,B 0,C 180,E1 10289.892,E2 10289.892} C_VEL
LIN {X 0,Y 393.666,Z 678.81,A -85,B 0,C 180,E1 10301.261,E2 10301.261} C_VEL
LIN {X 0,Y 393.591,Z 678.81,A -85,B 0,C 180,E1 10312.231,E2 10312.231} C_VEL
LIN {X 0,Y 394.015,Z 680.123,A -85,B 0,C 180,E1 10318.301,E2 10318.301} C_VEL
LIN {X 0,Y 411.147,Z 729.559,A -85,B 0,C 180,E1 10320.554,E2 10320.554} C_VEL
LIN {X 0,Y 407.793,Z 783.418,A -85,B 0,C 180,E1 10322.594,E2 10322.594} C_VEL
LIN {X 0,Y 402.484,Z 831.739,A -85,B 0,C 180,E1 10326.678,E2 10326.678} C_VEL
LIN {X 0,Y 398.137,Z 871.858,A -85,B 0,C 180,E1 10332.732,E2 10332.732} C_VEL
LIN {X 0,Y 396.344,Z 899.075,A -85,B 0,C 180,E1 10340.078,E2 10340.078} C_VEL
LIN {X 0,Y 396.315,Z 908.704,A -85,B 0,C 180,E1 10345.174,E2 10345.174} C_VEL
LIN {X 0,Y 388.416,Z 910.365,A -85,B 0,C 180,E1 10350.23,E2 10350.23} C_VEL
LIN {X 0,Y 388.102,Z 903.833,A -85,B 0,C 180,E1 10357.301,E2 10357.301} C_VEL
LIN {X 0,Y 389.017,Z 882.851,A -85,B 0,C 180,E1 10364.688,E2 10364.688} C_VEL
LIN {X 0,Y 392.59,Z 846.92,A -85,B 0,C 180,E1 10371.395,E2 10371.395} C_VEL
LIN {X 0,Y 397.694,Z 801.348,A -85,B 0,C 180,E1 10376.219,E2 10376.219} C_VEL
LIN {X 0,Y 402.013,Z 748.534,A -85,B 0,C 180,E1 10379.01,E2 10379.01} C_VEL
LIN {X 0,Y 400.012,Z 722.935,A -85,B 0,C 180,E1 10379.755,E2 10379.755} C_VEL
LIN {X 0,Y 385.691,Z 678.81,A -85,B 0,C 180,E1 10381.506,E2 10381.506} C_VEL
LIN {X 0,Y 385.536,Z 678.81,A -85,B 0,C 180,E1 10393.258,E2 10393.258} C_VEL
LIN {X 0,Y 385.48,Z 678.81,A -85,B 0,C 180,E1 10403.807,E2 10403.807} C_VEL
LIN {X 0,Y 385.767,Z 678.81,A -85,B 0,C 180,E1 10413.099,E2 10413.099} C_VEL
LIN {X 0,Y 386.196,Z 678.81,A -85,B 0,C 180,E1 10425.199,E2 10425.199} C_VEL
LIN {X 0,Y 387.027,Z 678.81,A -85,B 0,C 180,E1 10436.626,E2 10436.626} C_VEL
LIN {X 0,Y 386.705,Z 678.81,A -85,B 0,C 180,E1 10450.17,E2 10450.17} C_VEL
LIN {X 0,Y 386.27,Z 678.81,A -85,B 0,C 180,E1 10459.507,E2 10459.507} C_VEL
LIN {X 0,Y 385.83,Z 678.81,A -85,B 0,C 180,E1 10469.448,E2 10469.448} C_VEL
LIN {X 0,Y 385.492,Z 678.81,A -85,B 0,C 180,E1 10480.507,E2 10480.507} C_VEL
LIN {X 0,Y 385.455,Z 678.81,A -85,B 0,C 180,E1 10490.15,E2 10490.15} C_VEL
LIN {X 0,Y 385.671,Z 678.81,A -85,B 0,C 180,E1 10500.538,E2 10500.538} C_VEL
LIN {X 0,Y 385.89,Z 678.81,A -85,B 0,C 180,E1 10510.472,E2 10510.472} C_VEL
LIN {X 0,Y 386.763,Z 678.81,A -85,B 0,C 180,E1 10522.107,E2 10522.107} C_VEL
LIN {X 0,Y 387.358,Z 680.536,A -85,B 0,C 180,E1 10529.215,E2 10529.215} C_VEL
LIN {X 0,Y 396.839,Z 724.356,A -85,B 0,C 180,E1 10532.272,E2 10532.272} C_VEL
LIN {X 0,Y 393.044,Z 759.704,A -85,B 0,C 180,E1 10536.373,E2 10536.373} C_VEL
LIN {X 0,Y 390.305,Z 783.618,A -85,B 0,C 180,E1 10541.778,E2 10541.778} C_VEL
LIN {X 0,Y 389.141,Z 794.334,A -85,B 0,C 180,E1 10547.167,E2 10547.167} C_VEL
LIN {X 0,Y 389.543,Z 793.735,A -85,B 0,C 180,E1 10554.145,E2 10554.145} C_VEL
LIN {X 0,Y 392.075,Z 778.33,A -85,B 0,C 180,E1 10560.546,E2 10560.546} C_VEL
LIN {X 0,Y 396.119,Z 750.075,A -85,B 0,C 180,E1 10565.776,E2 10565.776} C_VEL
LIN {X 0,Y 397.483,Z 714.992,A -85,B 0,C 180,E1 10569.337,E2 10569.337} C_VEL
LIN {X 0,Y 385.661,Z 678.81,A -85,B 0,C 180,E1 10572.208,E2 10572.208} C_VEL
LIN {X 0,Y 385.436,Z 678.81,A -85,B 0,C 180,E1 10583.817,E2 10583.817} C_VEL
LIN {X 0,Y 385.773,Z 678.81,A -85,B 0,C 180,E1 10593.104,E2 10593.104} C_VEL
LIN {X 0,Y 386.187,Z 678.81,A -85,B 0,C 180,E1 10605.203,E2 10605.203} C_VEL
LIN {X 0,Y 387.027,Z 678.81,A -85,B 0,C 180,E1 10616.63,E2 10616.63} C_VEL
LIN {X 0,Y 386.848,Z 678.81,A -85,B 0,C 180,E1 10627.894,E2 10627.894} C_VEL
LIN {X 0,Y 386.229,Z 678.81,A -85,B 0,C 180,E1 10639.514,E2 10639.514} C_VEL
LIN {X 0,Y 385.876,Z 678.81,A -85,B 0,C 180,E1 10649.45,E2 10649.45} C_VEL
LIN {X 0,Y 385.658,Z 678.81,A -85,B 0,C 180,E1 10660.492,E2 10660.492} C_VEL
LIN {X 0,Y 385.584,Z 678.81,A -85,B 0,C 180,E1 10670.134,E2 10670.134} C_VEL
LIN {X 0,Y 386,Z 680.419,A -85,B 0,C 180,E1 10677.627,E2 10677.627} C_VEL
LIN {X 0,Y 403.971,Z 730.228,A -85,B 0,C 180,E1 10680.057,E2 10680.057} C_VEL
LIN {X 0,Y 400.343,Z 784.423,A -85,B 0,C 180,E1 10682.209,E2 10682.209} C_VEL
LIN {X 0,Y 394.613,Z 833.198,A -85,B 0,C 180,E1 10686.525,E2 10686.525} C_VEL
LIN {X 0,Y 390.158,Z 872.152,A -85,B 0,C 180,E1 10692.679,E2 10692.679} C_VEL
LIN {X 0,Y 388.392,Z 897.915,A -85,B 0,C 180,E1 10699.873,E2 10699.873} C_VEL
LIN {X 0,Y 388.311,Z 909.112,A -85,B 0,C 180,E1 10706.639,E2 10706.639} C_VEL
LIN {X 0,Y 388.416,Z 910.365,A -85,B 0,C 180,E1 10710.23,E2 10710.23} C_VEL
LIN {X 0,Y 380.357,Z 905.814,A -85,B 0,C 180,E1 10715.363,E2 10715.363} C_VEL
LIN {X 0,Y 380.406,Z 889.626,A -85,B 0,C 180,E1 10722.674,E2 10722.674} C_VEL
LIN {X 0,Y 383.037,Z 859.02,A -85,B 0,C 180,E1 10729.679,E2 10729.679} C_VEL
LIN {X 0,Y 388.211,Z 817.137,A -85,B 0,C 180,E1 10735.158,E2 10735.158} C_VEL
LIN {X 0,Y 393.323,Z 767.327,A -85,B 0,C 180,E1 10738.677,E2 10738.677} C_VEL
LIN {X 0,Y 393.092,Z 726.098,A -85,B 0,C 180,E1 10740.107,E2 10740.107} C_VEL
LIN {X 0,Y 377.635,Z 678.81,A -85,B 0,C 180,E1 10742.203,E2 10742.203} C_VEL
LIN {X 0,Y 377.425,Z 678.81,A -85,B 0,C 180,E1 10751.933,E2 10751.933} C_VEL
LIN {X 0,Y 377.445,Z 678.81,A -85,B 0,C 180,E1 10761.629,E2 10761.629} C_VEL
LIN {X 0,Y 377.741,Z 678.81,A -85,B 0,C 180,E1 10772.479,E2 10772.479} C_VEL
LIN {X 0,Y 378.008,Z 678.81,A -85,B 0,C 180,E1 10782.473,E2 10782.473} C_VEL
LIN {X 0,Y 378.766,Z 678.81,A -85,B 0,C 180,E1 10794.249,E2 10794.249} C_VEL
LIN {X 0,Y 378.408,Z 678.81,A -85,B 0,C 180,E1 10801.147,E2 10801.147} C_VEL
LIN {X 0,Y 378.545,Z 678.81,A -85,B 0,C 180,E1 10812.736,E2 10812.736} C_VEL
LIN {X 0,Y 378.122,Z 678.81,A -85,B 0,C 180,E1 10822.411,E2 10822.411} C_VEL
LIN {X 0,Y 377.564,Z 678.81,A -85,B 0,C 180,E1 10832.861,E2 10832.861} C_VEL
LIN {X 0,Y 377.375,Z 678.81,A -85,B 0,C 180,E1 10844.727,E2 10844.727} C_VEL
LIN {X 0,Y 377.459,Z 678.81,A -85,B 0,C 180,E1 10855.507,E2 10855.507} C_VEL
LIN {X 0,Y 377.663,Z 678.81,A -85,B 0,C 180,E1 10865.044,E2 10865.044} C_VEL
LIN {X 0,Y 378.162,Z 678.81,A -85,B 0,C 180,E1 10874.88,E2 10874.88} C_VEL
LIN {X 0,Y 379.023,Z 678.81,A -85,B 0,C 180,E1 10886.557,E2 10886.557} C_VEL
LIN {X 0,Y 379.523,Z 680.686,A -85,B 0,C 180,E1 10888.714,E2 10888.714} C_VEL
LIN {X 0,Y 389.38,Z 724.121,A -85,B 0,C 180,E1 10891.804,E2 10891.804} C_VEL
LIN {X 0,Y 385.48,Z 759.71,A -85,B 0,C 180,E1 10895.932,E2 10895.932} C_VEL
LIN {X 0,Y 382.501,Z 784.167,A -85,B 0,C 180,E1 10901.442,E2 10901.442} C_VEL
LIN {X 0,Y 381.209,Z 795.729,A -85,B 0,C 180,E1 10907.372,E2 10907.372} C_VEL
LIN {X 0,Y 381.458,Z 796.101,A -85,B 0,C 180,E1 10913.127,E2 10913.127} C_VEL
LIN {X 0,Y 383.756,Z 782.968,A -85,B 0,C 180,E1 10919.843,E2 10919.843} C_VEL
LIN {X 0,Y 387.727,Z 757.822,A -85,B 0,C 180,E1 10925.241,E2 10925.241} C_VEL
LIN {X 0,Y 390.906,Z 720.318,A -85,B 0,C 180,E1 10929.46,E2 10929.46} C_VEL
LIN {X 0,Y 377.57,Z 678.81,A -85,B 0,C 180,E1 10933.158,E2 10933.158} C_VEL
LIN {X 0,Y 377.462,Z 678.81,A -85,B 0,C 180,E1 10945.506,E2 10945.506} C_VEL
LIN {X 0,Y 377.741,Z 678.81,A -85,B 0,C 180,E1 10955.051,E2 10955.051} C_VEL
LIN {X 0,Y 378.167,Z 678.81,A -85,B 0,C 180,E1 10964.882,E2 10964.882} C_VEL
LIN {X 0,Y 379.006,Z 678.81,A -85,B 0,C 180,E1 10976.559,E2 10976.559} C_VEL
LIN {X 0,Y 378.811,Z 678.81,A -85,B 0,C 180,E1 10988.063,E2 10988.063} C_VEL
LIN {X 0,Y 378.158,Z 678.81,A -85,B 0,C 180,E1 10999.948,E2 10999.948} C_VEL
LIN {X 0,Y 377.759,Z 678.81,A -85,B 0,C 180,E1 11010.265,E2 11010.265} C_VEL
LIN {X 0,Y 377.531,Z 678.81,A -85,B 0,C 180,E1 11021.958,E2 11021.958} C_VEL
LIN {X 0,Y 377.539,Z 678.81,A -85,B 0,C 180,E1 11031.619,E2 11031.619} C_VEL
LIN {X 0,Y 377.957,Z 680.545,A -85,B 0,C 180,E1 11036.912,E2 11036.912} C_VEL
LIN {X 0,Y 396.871,Z 732.705,A -85,B 0,C 180,E1 11039.585,E2 11039.585} C_VEL
LIN {X 0,Y 392.825,Z 785.873,A -85,B 0,C 180,E1 11041.834,E2 11041.834} C_VEL
LIN {X 0,Y 386.843,Z 833.945,A -85,B 0,C 180,E1 11046.274,E2 11046.274} C_VEL
LIN {X 0,Y 382.155,Z 872.659,A -85,B 0,C 180,E1 11052.673,E2 11052.673} C_VEL
LIN {X 0,Y 380.387,Z 898.188,A -85,B 0,C 180,E1 11060.238,E2 11060.238} C_VEL
LIN {X 0,Y 380.381,Z 907.958,A -85,B 0,C 180,E1 11066.569,E2 11066.569} C_VEL
LIN {X 0,Y 380.469,Z 907.879,A -85,B 0,C 180,E1 11073.43,E2 11073.43} C_VEL
LIN {X 0,Y 380.357,Z 905.814,A -85,B 0,C 180,E1 11075.363,E2 11075.363} C_VEL
LIN {X 0,Y 372.407,Z 895.39,A -85,B 0,C 180,E1 11080.407,E2 11080.407} C_VEL
LIN {X 0,Y 374.167,Z 868.339,A -85,B 0,C 180,E1 11088.014,E2 11088.014} C_VEL
LIN {X 0,Y 379.1,Z 828.531,A -85,B 0,C 180,E1 11094.224,E2 11094.224} C_VEL
LIN {X 0,Y 384.686,Z 779.848,A -85,B 0,C 180,E1 11098.415,E2 11098.415} C_VEL
LIN {X 0,Y 386.047,Z 728.911,A -85,B 0,C 180,E1 11100.48,E2 11100.48} C_VEL
LIN {X 0,Y 369.576,Z 678.81,A -85,B 0,C 180,E1 11102.663,E2 11102.663} C_VEL
LIN {X 0,Y 369.338,Z 678.81,A -85,B 0,C 180,E1 11114.018,E2 11114.018} C_VEL
LIN {X 0,Y 369.371,Z 678.81,A -85,B 0,C 180,E1 11123.43,E2 11123.43} C_VEL
LIN {X 0,Y 369.711,Z 678.81,A -85,B 0,C 180,E1 11134.465,E2 11134.465} C_VEL
LIN {X 0,Y 370.121,Z 678.81,A -85,B 0,C 180,E1 11144.54,E2 11144.54} C_VEL
LIN {X 0,Y 371.001,Z 678.81,A -85,B 0,C 180,E1 11156.48,E2 11156.48} C_VEL
LIN {X 0,Y 370.561,Z 678.81,A -85,B 0,C 180,E1 11168.239,E2 11168.239} C_VEL
LIN {X 0,Y 370.282,Z 678.81,A -85,B 0,C 180,E1 11177.9,E2 11177.9} C_VEL
LIN {X 0,Y 369.787,Z 678.81,A -85,B 0,C 180,E1 11188.159,E2 11188.159} C_VEL
LIN {X 0,Y 369.299,Z 678.81,A -85,B 0,C 180,E1 11199.563,E2 11199.563} C_VEL
LIN {X 0,Y 369.269,Z 678.81,A -85,B 0,C 180,E1 11210.433,E2 11210.433} C_VEL
LIN {X 0,Y 369.613,Z 678.81,A -85,B 0,C 180,E1 11221.976,E2 11221.976} C_VEL
LIN {X 0,Y 369.944,Z 678.81,A -85,B 0,C 180,E1 11232.082,E2 11232.082} C_VEL
LIN {X 0,Y 370.689,Z 678.81,A -85,B 0,C 180,E1 11241.762,E2 11241.762} C_VEL
LIN {X 0,Y 371.46,Z 680.825,A -85,B 0,C 180,E1 11248.185,E2 11248.185} C_VEL
LIN {X 0,Y 381.442,Z 723.815,A -85,B 0,C 180,E1 11251.279,E2 11251.279} C_VEL
LIN {X 0,Y 377.963,Z 759.698,A -85,B 0,C 180,E1 11255.472,E2 11255.472} C_VEL
LIN {X 0,Y 374.75,Z 784.698,A -85,B 0,C 180,E1 11261.09,E2 11261.09} C_VEL
LIN {X 0,Y 373.245,Z 797.214,A -85,B 0,C 180,E1 11267.754,E2 11267.754} C_VEL
LIN {X 0,Y 374.016,Z 795.139,A -85,B 0,C 180,E1 11275.216,E2 11275.216} C_VEL
LIN {X 0,Y 377.099,Z 778.318,A -85,B 0,C 180,E1 11281.795,E2 11281.795} C_VEL
LIN {X 0,Y 381.907,Z 749.064,A -85,B 0,C 180,E1 11287.065,E2 11287.065} C_VEL
LIN {X 0,Y 383.111,Z 719.259,A -85,B 0,C 180,E1 11290.218,E2 11290.218} C_VEL
LIN {X 0,Y 369.481,Z 678.81,A -85,B 0,C 180,E1 11294.047,E2 11294.047} C_VEL
LIN {X 0,Y 369.467,Z 678.81,A -85,B 0,C 180,E1 11306.325,E2 11306.325} C_VEL
LIN {X 0,Y 369.766,Z 678.81,A -85,B 0,C 180,E1 11317.431,E2 11317.431} C_VEL
LIN {X 0,Y 370.5,Z 678.81,A -85,B 0,C 180,E1 11329.381,E2 11329.381} C_VEL
LIN {X 0,Y 371.452,Z 678.81,A -85,B 0,C 180,E1 11338.832,E2 11338.832} C_VEL
LIN {X 0,Y 370.61,Z 678.81,A -85,B 0,C 180,E1 11350.621,E2 11350.621} C_VEL
LIN {X 0,Y 370.064,Z 678.81,A -85,B 0,C 180,E1 11362.68,E2 11362.68} C_VEL
LIN {X 0,Y 369.643,Z 678.81,A -85,B 0,C 180,E1 11373.663,E2 11373.663} C_VEL
LIN {X 0,Y 369.422,Z 678.81,A -85,B 0,C 180,E1 11384.038,E2 11384.038} C_VEL
LIN {X 0,Y 369.879,Z 680.499,A -85,B 0,C 180,E1 11396.134,E2 11396.134} C_VEL
LIN {X 0,Y 389.695,Z 732.585,A -85,B 0,C 180,E1 11399.013,E2 11399.013} C_VEL
LIN {X 0,Y 385.573,Z 785.64,A -85,B 0,C 180,E1 11401.336,E2 11401.336} C_VEL
LIN {X 0,Y 379.307,Z 832.881,A -85,B 0,C 180,E1 11405.79,E2 11405.79} C_VEL
LIN {X 0,Y 374.258,Z 871.789,A -85,B 0,C 180,E1 11412.359,E2 11412.359} C_VEL
LIN {X 0,Y 372.435,Z 897.031,A -85,B 0,C 180,E1 11420.028,E2 11420.028} C_VEL
LIN {X 0,Y 372.484,Z 906.906,A -85,B 0,C 180,E1 11426.616,E2 11426.616} C_VEL
LIN {X 0,Y 372.554,Z 906.63,A -85,B 0,C 180,E1 11433.562,E2 11433.562} C_VEL
LIN {X 0,Y 372.407,Z 895.39,A -85,B 0,C 180,E1 11440.407,E2 11440.407} C_VEL
LIN {X 0,Y 365.331,Z 880.019,A -85,B 0,C 180,E1 11445.253,E2 11445.253} C_VEL
LIN {X 0,Y 369.23,Z 845.167,A -85,B 0,C 180,E1 11452.239,E2 11452.239} C_VEL
LIN {X 0,Y 374.885,Z 800.282,A -85,B 0,C 180,E1 11457.34,E2 11457.34} C_VEL
LIN {X 0,Y 379.711,Z 748.395,A -85,B 0,C 180,E1 11460.302,E2 11460.302} C_VEL
LIN {X 0,Y 376.905,Z 724.668,A -85,B 0,C 180,E1 11461.148,E2 11461.148} C_VEL
LIN {X 0,Y 361.542,Z 678.81,A -85,B 0,C 180,E1 11463.227,E2 11463.227} C_VEL
LIN {X 0,Y 361.332,Z 678.81,A -85,B 0,C 180,E1 11473.866,E2 11473.866} C_VEL
LIN {X 0,Y 361.359,Z 678.81,A -85,B 0,C 180,E1 11485.458,E2 11485.458} C_VEL
LIN {X 0,Y 361.659,Z 678.81,A -85,B 0,C 180,E1 11496.504,E2 11496.504} C_VEL
LIN {X 0,Y 362.197,Z 678.81,A -85,B 0,C 180,E1 11506.674,E2 11506.674} C_VEL
LIN {X 0,Y 363.274,Z 678.81,A -85,B 0,C 180,E1 11518.801,E2 11518.801} C_VEL
LIN {X 0,Y 362.627,Z 678.81,A -85,B 0,C 180,E1 11530.853,E2 11530.853} C_VEL
LIN {X 0,Y 362.092,Z 678.81,A -85,B 0,C 180,E1 11540.868,E2 11540.868} C_VEL
LIN {X 0,Y 361.543,Z 678.81,A -85,B 0,C 180,E1 11551.646,E2 11551.646} C_VEL
LIN {X 0,Y 361.294,Z 678.81,A -85,B 0,C 180,E1 11563.872,E2 11563.872} C_VEL
LIN {X 0,Y 361.319,Z 678.81,A -85,B 0,C 180,E1 11575.459,E2 11575.459} C_VEL
LIN {X 0,Y 361.605,Z 678.81,A -85,B 0,C 180,E1 11586.504,E2 11586.504} C_VEL
LIN {X 0,Y 362.175,Z 678.81,A -85,B 0,C 180,E1 11596.676,E2 11596.676} C_VEL
LIN {X 0,Y 363.282,Z 680.345,A -85,B 0,C 180,E1 11607.606,E2 11607.606} C_VEL
LIN {X 0,Y 373.739,Z 724.862,A -85,B 0,C 180,E1 11610.878,E2 11610.878} C_VEL
LIN {X 0,Y 370.185,Z 761.47,A -85,B 0,C 180,E1 11615.292,E2 11615.292} C_VEL
LIN {X 0,Y 366.738,Z 787.036,A -85,B 0,C 180,E1 11621.336,E2 11621.336} C_VEL
LIN {X 0,Y 365.301,Z 798.693,A -85,B 0,C 180,E1 11628.154,E2 11628.154} C_VEL
LIN {X 0,Y 366.266,Z 795.76,A -85,B 0,C 180,E1 11635.788,E2 11635.788} C_VEL
LIN {X 0,Y 369.602,Z 778.889,A -85,B 0,C 180,E1 11642.299,E2 11642.299} C_VEL
LIN {X 0,Y 374.868,Z 748.755,A -85,B 0,C 180,E1 11647.717,E2 11647.717} C_VEL
LIN {X 0,Y 375.749,Z 720.589,A -85,B 0,C 180,E1 11650.764,E2 11650.764} C_VEL
LIN {X 0,Y 361.375,Z 678.81,A -85,B 0,C 180,E1 11654.748,E2 11654.748} C_VEL
LIN {X 0,Y 361.326,Z 678.81,A -85,B 0,C 180,E1 11665.46,E2 11665.46} C_VEL
LIN {X 0,Y 361.654,Z 678.81,A -85,B 0,C 180,E1 11676.509,E2 11676.509} C_VEL
LIN {X 0,Y 362.191,Z 678.81,A -85,B 0,C 180,E1 11686.678,E2 11686.678} C_VEL
LIN {X 0,Y 363.435,Z 678.81,A -85,B 0,C 180,E1 11698.806,E2 11698.806} C_VEL
LIN {X 0,Y 362.588,Z 678.81,A -85,B 0,C 180,E1 11710.859,E2 11710.859} C_VEL
LIN {X 0,Y 362.046,Z 678.81,A -85,B 0,C 180,E1 11720.876,E2 11720.876} C_VEL
LIN {X 0,Y 361.655,Z 678.81,A -85,B 0,C 180,E1 11731.64,E2 11731.64} C_VEL
LIN {X 0,Y 361.416,Z 678.81,A -85,B 0,C 180,E1 11743.86,E2 11743.86} C_VEL
LIN {X 0,Y 361.68,Z 679.993,A -85,B 0,C 180,E1 11755.291,E2 11755.291} C_VEL
LIN {X 0,Y 382.749,Z 734.501,A -85,B 0,C 180,E1 11758.488,E2 11758.488} C_VEL
LIN {X 0,Y 378.191,Z 786.576,A -85,B 0,C 180,E1 11760.887,E2 11760.887} C_VEL
LIN {X 0,Y 371.5,Z 833.968,A -85,B 0,C 180,E1 11765.569,E2 11765.569} C_VEL
LIN {X 0,Y 366.329,Z 871.361,A -85,B 0,C 180,E1 11772.138,E2 11772.138} C_VEL
LIN {X 0,Y 364.479,Z 895.886,A -85,B 0,C 180,E1 11779.808,E2 11779.808} C_VEL
LIN {X 0,Y 364.559,Z 905.654,A -85,B 0,C 180,E1 11786.42,E2 11786.42} C_VEL
LIN {X 0,Y 364.633,Z 905.471,A -85,B 0,C 180,E1 11793.579,E2 11793.579} C_VEL
LIN {X 0,Y 364.371,Z 892.344,A -85,B 0,C 180,E1 11801.317,E2 11801.317} C_VEL
LIN {X 0,Y 365.331,Z 880.019,A -85,B 0,C 180,E1 11805.253,E2 11805.253} C_VEL
LIN {X 0,Y 359.038,Z 860.245,A -85,B 0,C 180,E1 11809.817,E2 11809.817} C_VEL
LIN {X 0,Y 364.763,Z 819.01,A -85,B 0,C 180,E1 11815.902,E2 11815.902} C_VEL
LIN {X 0,Y 370.749,Z 768.755,A -85,B 0,C 180,E1 11819.864,E2 11819.864} C_VEL
LIN {X 0,Y 370.937,Z 730.882,A -85,B 0,C 180,E1 11821.395,E2 11821.395} C_VEL
LIN {X 0,Y 353.455,Z 678.81,A -85,B 0,C 180,E1 11823.757,E2 11823.757} C_VEL
LIN {X 0,Y 353.288,Z 678.81,A -85,B 0,C 180,E1 11835.134,E2 11835.134} C_VEL
LIN {X 0,Y 353.36,Z 678.81,A -85,B 0,C 180,E1 11847.527,E2 11847.527} C_VEL
LIN {X 0,Y 353.69,Z 678.81,A -85,B 0,C 180,E1 11858.607,E2 11858.607} C_VEL
LIN {X 0,Y 354.407,Z 678.81,A -85,B 0,C 180,E1 11868.887,E2 11868.887} C_VEL
LIN {X 0,Y 355.267,Z 678.81,A -85,B 0,C 180,E1 11878.774,E2 11878.774} C_VEL
LIN {X 0,Y 354.576,Z 678.81,A -85,B 0,C 180,E1 11891.102,E2 11891.102} C_VEL
LIN {X 0,Y 353.919,Z 678.81,A -85,B 0,C 180,E1 11902.797,E2 11902.797} C_VEL
LIN {X 0,Y 353.36,Z 678.81,A -85,B 0,C 180,E1 11913.128,E2 11913.128} C_VEL
LIN {X 0,Y 353.219,Z 678.81,A -85,B 0,C 180,E1 11925.145,E2 11925.145} C_VEL
LIN {X 0,Y 353.318,Z 678.81,A -85,B 0,C 180,E1 11937.528,E2 11937.528} C_VEL
LIN {X 0,Y 353.632,Z 678.81,A -85,B 0,C 180,E1 11948.607,E2 11948.607} C_VEL
LIN {X 0,Y 354.401,Z 678.81,A -85,B 0,C 180,E1 11958.89,E2 11958.89} C_VEL
LIN {X 0,Y 355.266,Z 680.544,A -85,B 0,C 180,E1 11967.028,E2 11967.028} C_VEL
LIN {X 0,Y 365.755,Z 724.072,A -85,B 0,C 180,E1 11970.275,E2 11970.275} C_VEL
LIN {X 0,Y 362.963,Z 759.542,A -85,B 0,C 180,E1 11974.496,E2 11974.496} C_VEL
LIN {X 0,Y 359.259,Z 785.7,A -85,B 0,C 180,E1 11980.342,E2 11980.342} C_VEL
LIN {X 0,Y 357.488,Z 799.112,A -85,B 0,C 180,E1 11987.227,E2 11987.227} C_VEL
LIN {X 0,Y 358.042,Z 798.961,A -85,B 0,C 180,E1 11994.318,E2 11994.318} C_VEL
LIN {X 0,Y 361.148,Z 784.886,A -85,B 0,C 180,E1 12001.284,E2 12001.284} C_VEL
LIN {X 0,Y 366.306,Z 757.473,A -85,B 0,C 180,E1 12007.148,E2 12007.148} C_VEL
LIN {X 0,Y 368.954,Z 724.429,A -85,B 0,C 180,E1 12011.064,E2 12011.064} C_VEL
LIN {X 0,Y 354.989,Z 683.646,A -85,B 0,C 180,E1 12015.034,E2 12015.034} C_VEL
LIN {X 0,Y 353.323,Z 678.81,A -85,B 0,C 180,E1 12015.657,E2 12015.657} C_VEL
LIN {X 0,Y 353.339,Z 678.81,A -85,B 0,C 180,E1 12027.531,E2 12027.531} C_VEL
LIN {X 0,Y 353.686,Z 678.81,A -85,B 0,C 180,E1 12038.612,E2 12038.612} C_VEL
LIN {X 0,Y 354.404,Z 678.81,A -85,B 0,C 180,E1 12048.892,E2 12048.892} C_VEL
LIN {X 0,Y 355.441,Z 678.81,A -85,B 0,C 180,E1 12058.779,E2 12058.779} C_VEL
LIN {X 0,Y 354.54,Z 678.81,A -85,B 0,C 180,E1 12071.109,E2 12071.109} C_VEL
LIN {X 0,Y 353.909,Z 678.81,A -85,B 0,C 180,E1 12082.793,E2 12082.793} C_VEL
LIN {X 0,Y 353.488,Z 678.81,A -85,B 0,C 180,E1 12093.16,E2 12093.16} C_VEL
LIN {X 0,Y 353.341,Z 678.81,A -85,B 0,C 180,E1 12105.132,E2 12105.132} C_VEL
LIN {X 0,Y 353.696,Z 680.628,A -85,B 0,C 180,E1 12114.444,E2 12114.444} C_VEL
LIN {X 0,Y 375.541,Z 735.333,A -85,B 0,C 180,E1 12117.899,E2 12117.899} C_VEL
LIN {X 0,Y 370.832,Z 787.368,A -85,B 0,C 180,E1 12120.42,E2 12120.42} C_VEL
LIN {X 0,Y 363.884,Z 833.991,A -85,B 0,C 180,E1 12125.188,E2 12125.188} C_VEL
LIN {X 0,Y 358.359,Z 871.459,A -85,B 0,C 180,E1 12132.035,E2 12132.035} C_VEL
LIN {X 0,Y 356.498,Z 896.017,A -85,B 0,C 180,E1 12140.196,E2 12140.196} C_VEL
LIN {X 0,Y 356.828,Z 905.576,A -85,B 0,C 180,E1 12148.234,E2 12148.234} C_VEL
LIN {X 0,Y 356.444,Z 901.594,A -85,B 0,C 180,E1 12156.11,E2 12156.11} C_VEL
LIN {X 0,Y 356.839,Z 883.475,A -85,B 0,C 180,E1 12164.154,E2 12164.154} C_VEL
LIN {X 0,Y 359.038,Z 860.245,A -85,B 0,C 180,E1 12169.817,E2 12169.817} C_VEL
LIN {X 0,Y 354.683,Z 836.382,A -85,B 0,C 180,E1 12173.995,E2 12173.995} C_VEL
LIN {X 0,Y 360.806,Z 790.031,A -85,B 0,C 180,E1 12178.926,E2 12178.926} C_VEL
LIN {X 0,Y 364.926,Z 737.447,A -85,B 0,C 180,E1 12181.61,E2 12181.61} C_VEL
LIN {X 0,Y 345.362,Z 678.81,A -85,B 0,C 180,E1 12184.591,E2 12184.591} C_VEL
LIN {X 0,Y 345.17,Z 678.81,A -85,B 0,C 180,E1 12197.036,E2 12197.036} C_VEL
LIN {X 0,Y 345.336,Z 678.81,A -85,B 0,C 180,E1 12208.971,E2 12208.971} C_VEL
LIN {X 0,Y 345.764,Z 678.81,A -85,B 0,C 180,E1 12220.778,E2 12220.778} C_VEL
LIN {X 0,Y 346.568,Z 678.81,A -85,B 0,C 180,E1 12231.181,E2 12231.181} C_VEL
LIN {X 0,Y 346.394,Z 678.81,A -85,B 0,C 180,E1 12241.253,E2 12241.253} C_VEL
LIN {X 0,Y 346.535,Z 678.81,A -85,B 0,C 180,E1 12251.363,E2 12251.363} C_VEL
LIN {X 0,Y 345.949,Z 678.81,A -85,B 0,C 180,E1 12261.891,E2 12261.891} C_VEL
LIN {X 0,Y 345.335,Z 678.81,A -85,B 0,C 180,E1 12273.318,E2 12273.318} C_VEL
LIN {X 0,Y 345.117,Z 678.81,A -85,B 0,C 180,E1 12283.487,E2 12283.487} C_VEL
LIN {X 0,Y 345.266,Z 678.81,A -85,B 0,C 180,E1 12294.403,E2 12294.403} C_VEL
LIN {X 0,Y 345.494,Z 678.81,A -85,B 0,C 180,E1 12305.337,E2 12305.337} C_VEL
LIN {X 0,Y 346.11,Z 678.81,A -85,B 0,C 180,E1 12316.046,E2 12316.046} C_VEL
LIN {X 0,Y 347.07,Z 679.89,A -85,B 0,C 180,E1 12326.399,E2 12326.399} C_VEL
LIN {X 0,Y 357.49,Z 722.169,A -85,B 0,C 180,E1 12329.539,E2 12329.539} C_VEL
LIN {X 0,Y 356.681,Z 752.311,A -85,B 0,C 180,E1 12332.936,E2 12332.936} C_VEL
LIN {X 0,Y 352.398,Z 781.795,A -85,B 0,C 180,E1 12338.669,E2 12338.669} C_VEL
LIN {X 0,Y 349.94,Z 797.716,A -85,B 0,C 180,E1 12345.082,E2 12345.082} C_VEL
LIN {X 0,Y 349.592,Z 801.8,A -85,B 0,C 180,E1 12351.653,E2 12351.653} C_VEL
LIN {X 0,Y 351.778,Z 792.811,A -85,B 0,C 180,E1 12359.146,E2 12359.146} C_VEL
LIN {X 0,Y 356.789,Z 769.528,A -85,B 0,C 180,E1 12365.747,E2 12365.747} C_VEL
LIN {X 0,Y 362.794,Z 734.242,A -85,B 0,C 180,E1 12370.674,E2 12370.674} C_VEL
LIN {X 0,Y 352.448,Z 695.76,A -85,B 0,C 180,E1 12374.814,E2 12374.814} C_VEL
LIN {X 0,Y 345.283,Z 678.81,A -85,B 0,C 180,E1 12376.485,E2 12376.485} C_VEL
LIN {X 0,Y 345.321,Z 678.81,A -85,B 0,C 180,E1 12388.976,E2 12388.976} C_VEL
LIN {X 0,Y 345.754,Z 678.81,A -85,B 0,C 180,E1 12400.783,E2 12400.783} C_VEL
LIN {X 0,Y 346.567,Z 678.81,A -85,B 0,C 180,E1 12411.186,E2 12411.186} C_VEL
LIN {X 0,Y 347.023,Z 678.81,A -85,B 0,C 180,E1 12421.256,E2 12421.256} C_VEL
LIN {X 0,Y 346.507,Z 678.81,A -85,B 0,C 180,E1 12431.369,E2 12431.369} C_VEL
LIN {X 0,Y 345.923,Z 678.81,A -85,B 0,C 180,E1 12441.898,E2 12441.898} C_VEL
LIN {X 0,Y 345.468,Z 678.81,A -85,B 0,C 180,E1 12453.31,E2 12453.31} C_VEL
LIN {X 0,Y 345.25,Z 678.81,A -85,B 0,C 180,E1 12463.51,E2 12463.51} C_VEL
LIN {X 0,Y 345.537,Z 680.436,A -85,B 0,C 180,E1 12473.491,E2 12473.491} C_VEL
LIN {X 0,Y 367.976,Z 734.412,A -85,B 0,C 180,E1 12477.178,E2 12477.178} C_VEL
LIN {X 0,Y 363.784,Z 786.214,A -85,B 0,C 180,E1 12479.788,E2 12479.788} C_VEL
LIN {X 0,Y 356.462,Z 832.926,A -85,B 0,C 180,E1 12484.635,E2 12484.635} C_VEL
LIN {X 0,Y 350.51,Z 870.353,A -85,B 0,C 180,E1 12491.618,E2 12491.618} C_VEL
LIN {X 0,Y 348.538,Z 894.887,A -85,B 0,C 180,E1 12499.97,E2 12499.97} C_VEL
LIN {X 0,Y 348.711,Z 903.362,A -85,B 0,C 180,E1 12506.257,E2 12506.257} C_VEL
LIN {X 0,Y 348.788,Z 903.042,A -85,B 0,C 180,E1 12513.742,E2 12513.742} C_VEL
LIN {X 0,Y 348.457,Z 889.468,A -85,B 0,C 180,E1 12521.874,E2 12521.874} C_VEL
LIN {X 0,Y 350.857,Z 861.924,A -85,B 0,C 180,E1 12529.585,E2 12529.585} C_VEL
LIN {X 0,Y 354.683,Z 836.382,A -85,B 0,C 180,E1 12533.995,E2 12533.995} C_VEL
LIN {X 0,Y 350.767,Z 809.114,A -85,B 0,C 180,E1 12537.628,E2 12537.628} C_VEL
LIN {X 0,Y 356.78,Z 757.904,A -85,B 0,C 180,E1 12541.312,E2 12541.312} C_VEL
LIN {X 0,Y 355.567,Z 732.014,A -85,B 0,C 180,E1 12542.419,E2 12542.419} C_VEL
LIN {X 0,Y 337.35,Z 678.81,A -85,B 0,C 180,E1 12545.063,E2 12545.063} C_VEL
LIN {X 0,Y 337.092,Z 678.81,A -85,B 0,C 180,E1 12555.743,E2 12555.743} C_VEL
LIN {X 0,Y 337.303,Z 678.81,A -85,B 0,C 180,E1 12566.338,E2 12566.338} C_VEL
LIN {X 0,Y 337.574,Z 678.81,A -85,B 0,C 180,E1 12577.531,E2 12577.531} C_VEL
LIN {X 0,Y 338.293,Z 678.81,A -85,B 0,C 180,E1 12588.351,E2 12588.351} C_VEL
LIN {X 0,Y 339.263,Z 678.81,A -85,B 0,C 180,E1 12598.716,E2 12598.716} C_VEL
LIN {X 0,Y 338.483,Z 678.81,A -85,B 0,C 180,E1 12611.637,E2 12611.637} C_VEL
LIN {X 0,Y 337.802,Z 678.81,A -85,B 0,C 180,E1 12622.936,E2 12622.936} C_VEL
LIN {X 0,Y 337.28,Z 678.81,A -85,B 0,C 180,E1 12634.222,E2 12634.222} C_VEL
LIN {X 0,Y 337.028,Z 678.81,A -85,B 0,C 180,E1 12645.74,E2 12645.74} C_VEL
LIN {X 0,Y 337.24,Z 678.81,A -85,B 0,C 180,E1 12656.355,E2 12656.355} C_VEL
LIN {X 0,Y 337.52,Z 678.81,A -85,B 0,C 180,E1 12667.532,E2 12667.532} C_VEL
LIN {X 0,Y 338.284,Z 678.81,A -85,B 0,C 180,E1 12678.354,E2 12678.354} C_VEL
LIN {X 0,Y 339.045,Z 680.575,A -85,B 0,C 180,E1 12685.789,E2 12685.789} C_VEL
LIN {X 0,Y 349.608,Z 721.669,A -85,B 0,C 180,E1 12688.923,E2 12688.923} C_VEL
LIN {X 0,Y 349.84,Z 747.334,A -85,B 0,C 180,E1 12691.75,E2 12691.75} C_VEL
LIN {X 0,Y 345.169,Z 779.291,A -85,B 0,C 180,E1 12697.475,E2 12697.475} C_VEL
LIN {X 0,Y 342.279,Z 797.441,A -85,B 0,C 180,E1 12704.114,E2 12704.114} C_VEL
LIN {X 0,Y 341.76,Z 802.852,A -85,B 0,C 180,E1 12712.175,E2 12712.175} C_VEL
LIN {X 0,Y 344.257,Z 793.37,A -85,B 0,C 180,E1 12719.73,E2 12719.73} C_VEL
LIN {X 0,Y 349.694,Z 769.552,A -85,B 0,C 180,E1 12726.449,E2 12726.449} C_VEL
LIN {X 0,Y 355.57,Z 733.377,A -85,B 0,C 180,E1 12731.508,E2 12731.508} C_VEL
LIN {X 0,Y 343.543,Z 693.234,A -85,B 0,C 180,E1 12735.989,E2 12735.989} C_VEL
LIN {X 0,Y 337.145,Z 678.81,A -85,B 0,C 180,E1 12737.501,E2 12737.501} C_VEL
LIN {X 0,Y 337.31,Z 678.81,A -85,B 0,C 180,E1 12748.844,E2 12748.844} C_VEL
LIN {X 0,Y 337.702,Z 678.81,A -85,B 0,C 180,E1 12760.306,E2 12760.306} C_VEL
LIN {X 0,Y 338.549,Z 678.81,A -85,B 0,C 180,E1 12770.976,E2 12770.976} C_VEL
LIN {X 0,Y 339.029,Z 678.81,A -85,B 0,C 180,E1 12781.285,E2 12781.285} C_VEL
LIN {X 0,Y 338.457,Z 678.81,A -85,B 0,C 180,E1 12791.644,E2 12791.644} C_VEL
LIN {X 0,Y 337.787,Z 678.81,A -85,B 0,C 180,E1 12802.929,E2 12802.929} C_VEL
LIN {X 0,Y 337.397,Z 678.81,A -85,B 0,C 180,E1 12814.215,E2 12814.215} C_VEL
LIN {X 0,Y 337.153,Z 678.81,A -85,B 0,C 180,E1 12825.76,E2 12825.76} C_VEL
LIN {X 0,Y 337.466,Z 680.179,A -85,B 0,C 180,E1 12832.489,E2 12832.489} C_VEL
LIN {X 0,Y 360.852,Z 735.474,A -85,B 0,C 180,E1 12836.53,E2 12836.53} C_VEL
LIN {X 0,Y 356.506,Z 787.188,A -85,B 0,C 180,E1 12839.282,E2 12839.282} C_VEL
LIN {X 0,Y 348.686,Z 834.034,A -85,B 0,C 180,E1 12844.374,E2 12844.374} C_VEL
LIN {X 0,Y 342.511,Z 871.03,A -85,B 0,C 180,E1 12851.632,E2 12851.632} C_VEL
LIN {X 0,Y 340.545,Z 895.011,A -85,B 0,C 180,E1 12860.38,E2 12860.38} C_VEL
LIN {X 0,Y 341.112,Z 903.372,A -85,B 0,C 180,E1 12868.725,E2 12868.725} C_VEL
LIN {X 0,Y 340.559,Z 899.06,A -85,B 0,C 180,E1 12876.396,E2 12876.396} C_VEL
LIN {X 0,Y 341.148,Z 880.556,A -85,B 0,C 180,E1 12884.82,E2 12884.82} C_VEL
LIN {X 0,Y 345.173,Z 847.655,A -85,B 0,C 180,E1 12892.442,E2 12892.442} C_VEL
LIN {X 0,Y 350.767,Z 809.114,A -85,B 0,C 180,E1 12897.628,E2 12897.628} C_VEL
LIN {X 0,Y 347.228,Z 778.831,A -85,B 0,C 180,E1 12900.599,E2 12900.599} C_VEL
LIN {X 0,Y 348.847,Z 735.979,A -85,B 0,C 180,E1 12902.773,E2 12902.773} C_VEL
LIN {X 0,Y 329.337,Z 678.81,A -85,B 0,C 180,E1 12905.876,E2 12905.876} C_VEL
LIN {X 0,Y 329.069,Z 678.81,A -85,B 0,C 180,E1 12918.028,E2 12918.028} C_VEL
LIN {X 0,Y 329.291,Z 678.81,A -85,B 0,C 180,E1 12928.493,E2 12928.493} C_VEL
LIN {X 0,Y 329.701,Z 678.81,A -85,B 0,C 180,E1 12940.66,E2 12940.66} C_VEL
LIN {X 0,Y 330.63,Z 678.81,A -85,B 0,C 180,E1 12953.408,E2 12953.408} C_VEL
LIN {X 0,Y 330.388,Z 678.81,A -85,B 0,C 180,E1 12961.313,E2 12961.313} C_VEL
LIN {X 0,Y 330.43,Z 678.81,A -85,B 0,C 180,E1 12971.925,E2 12971.925} C_VEL
LIN {X 0,Y 329.801,Z 678.81,A -85,B 0,C 180,E1 12983.023,E2 12983.023} C_VEL
LIN {X 0,Y 329.115,Z 678.81,A -85,B 0,C 180,E1 12995.195,E2 12995.195} C_VEL
LIN {X 0,Y 329.022,Z 678.81,A -85,B 0,C 180,E1 13005.635,E2 13005.635} C_VEL
LIN {X 0,Y 329.245,Z 678.81,A -85,B 0,C 180,E1 13018.506,E2 13018.506} C_VEL
LIN {X 0,Y 329.664,Z 678.81,A -85,B 0,C 180,E1 13030.68,E2 13030.68} C_VEL
LIN {X 0,Y 330.636,Z 678.81,A -85,B 0,C 180,E1 13043.411,E2 13043.411} C_VEL
LIN {X 0,Y 330.919,Z 680.313,A -85,B 0,C 180,E1 13045.109,E2 13045.109} C_VEL
LIN {X 0,Y 341.62,Z 720.23,A -85,B 0,C 180,E1 13048.201,E2 13048.201} C_VEL
LIN {X 0,Y 342.511,Z 746.432,A -85,B 0,C 180,E1 13051.111,E2 13051.111} C_VEL
LIN {X 0,Y 337.573,Z 778.873,A -85,B 0,C 180,E1 13056.826,E2 13056.826} C_VEL
LIN {X 0,Y 334.5,Z 797.732,A -85,B 0,C 180,E1 13063.55,E2 13063.55} C_VEL
LIN {X 0,Y 333.731,Z 804.221,A -85,B 0,C 180,E1 13071.222,E2 13071.222} C_VEL
LIN {X 0,Y 335.997,Z 796.7,A -85,B 0,C 180,E1 13079.047,E2 13079.047} C_VEL
LIN {X 0,Y 341.394,Z 774.746,A -85,B 0,C 180,E1 13086.112,E2 13086.112} C_VEL
LIN {X 0,Y 348.34,Z 739.892,A -85,B 0,C 180,E1 13091.507,E2 13091.507} C_VEL
LIN {X 0,Y 340.137,Z 704.029,A -85,B 0,C 180,E1 13095.804,E2 13095.804} C_VEL
LIN {X 0,Y 329.084,Z 678.81,A -85,B 0,C 180,E1 13098.851,E2 13098.851} C_VEL
LIN {X 0,Y 329.346,Z 678.81,A -85,B 0,C 180,E1 13111.067,E2 13111.067} C_VEL
LIN {X 0,Y 329.79,Z 678.81,A -85,B 0,C 180,E1 13122.598,E2 13122.598} C_VEL
LIN {X 0,Y 330.63,Z 678.81,A -85,B 0,C 180,E1 13133.413,E2 13133.413} C_VEL
LIN {X 0,Y 331.021,Z 678.81,A -85,B 0,C 180,E1 13141.316,E2 13141.316} C_VEL
LIN {X 0,Y 330.406,Z 678.81,A -85,B 0,C 180,E1 13151.931,E2 13151.931} C_VEL
LIN {X 0,Y 329.785,Z 678.81,A -85,B 0,C 180,E1 13163.03,E2 13163.03} C_VEL
LIN {X 0,Y 329.249,Z 678.81,A -85,B 0,C 180,E1 13175.185,E2 13175.185} C_VEL
LIN {X 0,Y 329.145,Z 678.81,A -85,B 0,C 180,E1 13185.621,E2 13185.621} C_VEL
LIN {X 0,Y 329.362,Z 680.114,A -85,B 0,C 180,E1 13191.41,E2 13191.41} C_VEL
LIN {X 0,Y 353.399,Z 735.06,A -85,B 0,C 180,E1 13195.763,E2 13195.763} C_VEL
LIN {X 0,Y 351.414,Z 774.678,A -85,B 0,C 180,E1 13197.788,E2 13197.788} C_VEL
LIN {X 0,Y 343.261,Z 822.806,A -85,B 0,C 180,E1 13202.341,E2 13202.341} C_VEL
LIN {X 0,Y 335.751,Z 861.824,A -85,B 0,C 180,E1 13209.149,E2 13209.149} C_VEL
LIN {X 0,Y 332.628,Z 888.507,A -85,B 0,C 180,E1 13217.484,E2 13217.484} C_VEL
LIN {X 0,Y 332.85,Z 901.072,A -85,B 0,C 180,E1 13226.078,E2 13226.078} C_VEL
LIN {X 0,Y 332.911,Z 900.601,A -85,B 0,C 180,E1 13233.921,E2 13233.921} C_VEL
LIN {X 0,Y 332.552,Z 886.479,A -85,B 0,C 180,E1 13242.519,E2 13242.519} C_VEL
LIN {X 0,Y 335.421,Z 858.461,A -85,B 0,C 180,E1 13250.526,E2 13250.526} C_VEL
LIN {X 0,Y 341.83,Z 817.489,A -85,B 0,C 180,E1 13257.068,E2 13257.068} C_VEL
LIN {X 0,Y 347.228,Z 778.831,A -85,B 0,C 180,E1 13260.599,E2 13260.599} C_VEL
LIN {X 0,Y 342.965,Z 746.203,A -85,B 0,C 180,E1 13262.807,E2 13262.807} C_VEL
LIN {X 0,Y 321.199,Z 678.81,A -85,B 0,C 180,E1 13266.703,E2 13266.703} C_VEL
LIN {X 0,Y 321.007,Z 678.81,A -85,B 0,C 180,E1 13277.118,E2 13277.118} C_VEL
LIN {X 0,Y 321.108,Z 678.81,A -85,B 0,C 180,E1 13287.073,E2 13287.073} C_VEL
LIN {X 0,Y 321.549,Z 678.81,A -85,B 0,C 180,E1 13299.266,E2 13299.266} C_VEL
LIN {X 0,Y 322.45,Z 678.81,A -85,B 0,C 180,E1 13310.516,E2 13310.516} C_VEL
LIN {X 0,Y 322.373,Z 678.81,A -85,B 0,C 180,E1 13321.346,E2 13321.346} C_VEL
LIN {X 0,Y 322.377,Z 678.81,A -85,B 0,C 180,E1 13332.228,E2 13332.228} C_VEL
LIN {X 0,Y 321.686,Z 678.81,A -85,B 0,C 180,E1 13343.638,E2 13343.638} C_VEL
LIN {X 0,Y 321.073,Z 678.81,A -85,B 0,C 180,E1 13356.213,E2 13356.213} C_VEL
LIN {X 0,Y 320.949,Z 678.81,A -85,B 0,C 180,E1 13367.128,E2 13367.128} C_VEL
LIN {X 0,Y 321.064,Z 678.81,A -85,B 0,C 180,E1 13377.074,E2 13377.074} C_VEL
LIN {X 0,Y 321.507,Z 678.81,A -85,B 0,C 180,E1 13389.267,E2 13389.267} C_VEL
LIN {X 0,Y 322.47,Z 678.81,A -85,B 0,C 180,E1 13400.52,E2 13400.52} C_VEL
LIN {X 0,Y 322.922,Z 680.725,A -85,B 0,C 180,E1 13404.434,E2 13404.434} C_VEL
LIN {X 0,Y 333.697,Z 719.138,A -85,B 0,C 180,E1 13407.489,E2 13407.489} C_VEL
LIN {X 0,Y 335.163,Z 745.95,A -85,B 0,C 180,E1 13410.501,E2 13410.501} C_VEL
LIN {X 0,Y 329.927,Z 778.838,A -85,B 0,C 180,E1 13416.272,E2 13416.272} C_VEL
LIN {X 0,Y 326.671,Z 798.429,A -85,B 0,C 180,E1 13423.204,E2 13423.204} C_VEL
LIN {X 0,Y 325.74,Z 805.365,A -85,B 0,C 180,E1 13430.451,E2 13430.451} C_VEL
LIN {X 0,Y 327.75,Z 799.883,A -85,B 0,C 180,E1 13438.23,E2 13438.23} C_VEL
LIN {X 0,Y 332.952,Z 780.461,A -85,B 0,C 180,E1 13445.52,E2 13445.52} C_VEL
LIN {X 0,Y 340.409,Z 747.447,A -85,B 0,C 180,E1 13451.37,E2 13451.37} C_VEL
LIN {X 0,Y 338.467,Z 722.471,A -85,B 0,C 180,E1 13454.561,E2 13454.561} C_VEL
LIN {X 0,Y 321.009,Z 678.81,A -85,B 0,C 180,E1 13459.844,E2 13459.844} C_VEL
LIN {X 0,Y 321.333,Z 678.81,A -85,B 0,C 180,E1 13470.891,E2 13470.891} C_VEL
LIN {X 0,Y 321.751,Z 678.81,A -85,B 0,C 180,E1 13482.149,E2 13482.149} C_VEL
LIN {X 0,Y 322.602,Z 678.81,A -85,B 0,C 180,E1 13493.249,E2 13493.249} C_VEL
LIN {X 0,Y 323.027,Z 678.81,A -85,B 0,C 180,E1 13501.349,E2 13501.349} C_VEL
LIN {X 0,Y 322.352,Z 678.81,A -85,B 0,C 180,E1 13512.234,E2 13512.234} C_VEL
LIN {X 0,Y 321.675,Z 678.81,A -85,B 0,C 180,E1 13523.645,E2 13523.645} C_VEL
LIN {X 0,Y 321.217,Z 678.81,A -85,B 0,C 180,E1 13536.202,E2 13536.202} C_VEL
LIN {X 0,Y 321.086,Z 678.81,A -85,B 0,C 180,E1 13547.11,E2 13547.11} C_VEL
LIN {X 0,Y 321.251,Z 680.02,A -85,B 0,C 180,E1 13550.246,E2 13550.246} C_VEL
LIN {X 0,Y 345.93,Z 734.535,A -85,B 0,C 180,E1 13554.936,E2 13554.936} C_VEL
LIN {X 0,Y 346.714,Z 757.105,A -85,B 0,C 180,E1 13556.121,E2 13556.121} C_VEL
LIN {X 0,Y 338.851,Z 807.178,A -85,B 0,C 180,E1 13559.932,E2 13559.932} C_VEL
LIN {X 0,Y 330.222,Z 850.02,A -85,B 0,C 180,E1 13566.29,E2 13566.29} C_VEL
LIN {X 0,Y 325.231,Z 880.712,A -85,B 0,C 180,E1 13574.468,E2 13574.468} C_VEL
LIN {X 0,Y 324.694,Z 897.552,A -85,B 0,C 180,E1 13583.29,E2 13583.29} C_VEL
LIN {X 0,Y 325.095,Z 900.833,A -85,B 0,C 180,E1 13591.337,E2 13591.337} C_VEL
LIN {X 0,Y 324.643,Z 890.765,A -85,B 0,C 180,E1 13600.269,E2 13600.269} C_VEL
LIN {X 0,Y 326.525,Z 865.523,A -85,B 0,C 180,E1 13608.985,E2 13608.985} C_VEL
LIN {X 0,Y 332.436,Z 828.424,A -85,B 0,C 180,E1 13615.99,E2 13615.99} C_VEL
LIN {X 0,Y 339.495,Z 780.64,A -85,B 0,C 180,E1 13620.934,E2 13620.934} C_VEL
LIN {X 0,Y 342.965,Z 746.203,A -85,B 0,C 180,E1 13622.807,E2 13622.807} C_VEL
LIN {X 0,Y 336.714,Z 731.216,A -85,B 0,C 180,E1 13623.833,E2 13623.833} C_VEL
LIN {X 0,Y 327.244,Z 716.753,A -85,B 0,C 180,E1 13624.966,E2 13624.966} C_VEL
LIN {X 0,Y 313.144,Z 678.81,A -85,B 0,C 180,E1 13627.284,E2 13627.284} C_VEL
LIN {X 0,Y 312.889,Z 678.81,A -85,B 0,C 180,E1 13639.092,E2 13639.092} C_VEL
LIN {X 0,Y 313.139,Z 678.81,A -85,B 0,C 180,E1 13649.407,E2 13649.407} C_VEL
LIN {X 0,Y 313.668,Z 678.81,A -85,B 0,C 180,E1 13661.667,E2 13661.667} C_VEL
LIN {X 0,Y 314.567,Z 678.81,A -85,B 0,C 180,E1 13673.07,E2 13673.07} C_VEL
LIN {X 0,Y 314.358,Z 678.81,A -85,B 0,C 180,E1 13681.38,E2 13681.38} C_VEL
LIN {X 0,Y 314.321,Z 678.81,A -85,B 0,C 180,E1 13692.546,E2 13692.546} C_VEL
LIN {X 0,Y 313.576,Z 678.81,A -85,B 0,C 180,E1 13704.288,E2 13704.288} C_VEL
LIN {X 0,Y 312.977,Z 678.81,A -85,B 0,C 180,E1 13717.306,E2 13717.306} C_VEL
LIN {X 0,Y 312.838,Z 678.81,A -85,B 0,C 180,E1 13729.09,E2 13729.09} C_VEL
LIN {X 0,Y 313.092,Z 678.81,A -85,B 0,C 180,E1 13739.407,E2 13739.407} C_VEL
LIN {X 0,Y 313.632,Z 678.81,A -85,B 0,C 180,E1 13751.669,E2 13751.669} C_VEL
LIN {X 0,Y 314.841,Z 680.487,A -85,B 0,C 180,E1 13763.698,E2 13763.698} C_VEL
LIN {X 0,Y 326.187,Z 719.946,A -85,B 0,C 180,E1 13766.937,E2 13766.937} C_VEL
LIN {X 0,Y 327.543,Z 747.784,A -85,B 0,C 180,E1 13770.166,E2 13770.166} C_VEL
LIN {X 0,Y 322.129,Z 780.341,A -85,B 0,C 180,E1 13776.085,E2 13776.085} C_VEL
LIN {X 0,Y 318.597,Z 800.826,A -85,B 0,C 180,E1 13783.835,E2 13783.835} C_VEL
LIN {X 0,Y 317.94,Z 806.582,A -85,B 0,C 180,E1 13791.448,E2 13791.448} C_VEL
LIN {X 0,Y 320.647,Z 798.932,A -85,B 0,C 180,E1 13799.798,E2 13799.798} C_VEL
LIN {X 0,Y 327.026,Z 776.266,A -85,B 0,C 180,E1 13807.34,E2 13807.34} C_VEL
LIN {X 0,Y 334.53,Z 740.987,A -85,B 0,C 180,E1 13812.96,E2 13812.96} C_VEL
LIN {X 0,Y 323.849,Z 702.037,A -85,B 0,C 180,E1 13818.107,E2 13818.107} C_VEL
LIN {X 0,Y 313,Z 678.81,A -85,B 0,C 180,E1 13820.813,E2 13820.813} C_VEL
LIN {X 0,Y 313.34,Z 678.81,A -85,B 0,C 180,E1 13833.634,E2 13833.634} C_VEL
LIN {X 0,Y 313.891,Z 678.81,A -85,B 0,C 180,E1 13844.581,E2 13844.581} C_VEL
LIN {X 0,Y 314.837,Z 678.81,A -85,B 0,C 180,E1 13855.856,E2 13855.856} C_VEL
LIN {X 0,Y 314.739,Z 678.81,A -85,B 0,C 180,E1 13866.926,E2 13866.926} C_VEL
LIN {X 0,Y 313.824,Z 678.81,A -85,B 0,C 180,E1 13879.446,E2 13879.446} C_VEL
LIN {X 0,Y 313.204,Z 678.81,A -85,B 0,C 180,E1 13892.014,E2 13892.014} C_VEL
LIN {X 0,Y 312.966,Z 678.81,A -85,B 0,C 180,E1 13904.683,E2 13904.683} C_VEL
LIN {X 0,Y 313.36,Z 680.836,A -85,B 0,C 180,E1 13909.061,E2 13909.061} C_VEL
LIN {X 0,Y 338.185,Z 733.273,A -85,B 0,C 180,E1 13913.997,E2 13913.997} C_VEL
LIN {X 0,Y 340.491,Z 752.613,A -85,B 0,C 180,E1 13915.194,E2 13915.194} C_VEL
LIN {X 0,Y 332.418,Z 803.286,A -85,B 0,C 180,E1 13918.906,E2 13918.906} C_VEL
LIN {X 0,Y 323.515,Z 845.668,A -85,B 0,C 180,E1 13925.028,E2 13925.028} C_VEL
LIN {X 0,Y 317.686,Z 878.151,A -85,B 0,C 180,E1 13933.513,E2 13933.513} C_VEL
LIN {X 0,Y 316.724,Z 896.418,A -85,B 0,C 180,E1 13943.12,E2 13943.12} C_VEL
LIN {X 0,Y 317.171,Z 899.625,A -85,B 0,C 180,E1 13951.371,E2 13951.371} C_VEL
LIN {X 0,Y 316.742,Z 890.976,A -85,B 0,C 180,E1 13959.653,E2 13959.653} C_VEL
LIN {X 0,Y 318.254,Z 867.785,A -85,B 0,C 180,E1 13968.415,E2 13968.415} C_VEL
LIN {X 0,Y 324.186,Z 831.429,A -85,B 0,C 180,E1 13975.844,E2 13975.844} C_VEL
LIN {X 0,Y 331.256,Z 785.716,A -85,B 0,C 180,E1 13981.023,E2 13981.023} C_VEL
LIN {X 0,Y 334.228,Z 739.472,A -85,B 0,C 180,E1 13983.741,E2 13983.741} C_VEL
LIN {X 0,Y 327.244,Z 716.753,A -85,B 0,C 180,E1 13984.966,E2 13984.966} C_VEL
LIN {X 0,Y 308.874,Z 689.05,A -85,B 0,C 180,E1 13987.268,E2 13987.268} C_VEL
LIN {X 0,Y 304.986,Z 678.81,A -85,B 0,C 180,E1 13988.076,E2 13988.076} C_VEL
LIN {X 0,Y 304.819,Z 678.81,A -85,B 0,C 180,E1 14001.508,E2 14001.508} C_VEL
LIN {X 0,Y 305.184,Z 678.81,A -85,B 0,C 180,E1 14011.805,E2 14011.805} C_VEL
LIN {X 0,Y 305.817,Z 678.81,A -85,B 0,C 180,E1 14024.158,E2 14024.158} C_VEL
LIN {X 0,Y 306.82,Z 678.81,A -85,B 0,C 180,E1 14035.742,E2 14035.742} C_VEL
LIN {X 0,Y 306.384,Z 678.81,A -85,B 0,C 180,E1 14049.981,E2 14049.981} C_VEL
LIN {X 0,Y 305.714,Z 678.81,A -85,B 0,C 180,E1 14061.855,E2 14061.855} C_VEL
LIN {X 0,Y 304.995,Z 678.81,A -85,B 0,C 180,E1 14074.902,E2 14074.902} C_VEL
LIN {X 0,Y 304.727,Z 678.81,A -85,B 0,C 180,E1 14087.755,E2 14087.755} C_VEL
LIN {X 0,Y 305.056,Z 678.81,A -85,B 0,C 180,E1 14100.524,E2 14100.524} C_VEL
LIN {X 0,Y 305.585,Z 678.81,A -85,B 0,C 180,E1 14111.168,E2 14111.168} C_VEL
LIN {X 0,Y 306.621,Z 679.769,A -85,B 0,C 180,E1 14122.893,E2 14122.893} C_VEL
LIN {X 0,Y 318.681,Z 720.816,A -85,B 0,C 180,E1 14126.375,E2 14126.375} C_VEL
LIN {X 0,Y 320.07,Z 748.624,A -85,B 0,C 180,E1 14129.683,E2 14129.683} C_VEL
LIN {X 0,Y 314.337,Z 781.842,A -85,B 0,C 180,E1 14135.888,E2 14135.888} C_VEL
LIN {X 0,Y 310.793,Z 801.42,A -85,B 0,C 180,E1 14143.411,E2 14143.411} C_VEL
LIN {X 0,Y 310.062,Z 807.761,A -85,B 0,C 180,E1 14151.535,E2 14151.535} C_VEL
LIN {X 0,Y 312.603,Z 801.378,A -85,B 0,C 180,E1 14159.465,E2 14159.465} C_VEL
LIN {X 0,Y 318.82,Z 780.738,A -85,B 0,C 180,E1 14167.118,E2 14167.118} C_VEL
LIN {X 0,Y 326.851,Z 748.26,A -85,B 0,C 180,E1 14172.884,E2 14172.884} C_VEL
LIN {X 0,Y 321.34,Z 715.428,A -85,B 0,C 180,E1 14177.476,E2 14177.476} C_VEL
LIN {X 0,Y 304.991,Z 678.81,A -85,B 0,C 180,E1 14182.48,E2 14182.48} C_VEL
LIN {X 0,Y 305.305,Z 678.81,A -85,B 0,C 180,E1 14195.009,E2 14195.009} C_VEL
LIN {X 0,Y 306.049,Z 678.81,A -85,B 0,C 180,E1 14207.109,E2 14207.109} C_VEL
LIN {X 0,Y 307.328,Z 678.81,A -85,B 0,C 180,E1 14218.588,E2 14218.588} C_VEL
LIN {X 0,Y 306.477,Z 678.81,A -85,B 0,C 180,E1 14229.984,E2 14229.984} C_VEL
LIN {X 0,Y 305.658,Z 678.81,A -85,B 0,C 180,E1 14241.866,E2 14241.866} C_VEL
LIN {X 0,Y 305.131,Z 678.81,A -85,B 0,C 180,E1 14254.892,E2 14254.892} C_VEL
LIN {X 0,Y 305.067,Z 680.444,A -85,B 0,C 180,E1 14267.656,E2 14267.656} C_VEL
LIN {X 0,Y 330.592,Z 732.611,A -85,B 0,C 180,E1 14273.045,E2 14273.045} C_VEL
LIN {X 0,Y 333.837,Z 752.549,A -85,B 0,C 180,E1 14274.438,E2 14274.438} C_VEL
LIN {X 0,Y 325.483,Z 802.48,A -85,B 0,C 180,E1 14278.167,E2 14278.167} C_VEL
LIN {X 0,Y 316.127,Z 844.699,A -85,B 0,C 180,E1 14284.403,E2 14284.403} C_VEL
LIN {X 0,Y 309.992,Z 876.502,A -85,B 0,C 180,E1 14292.854,E2 14292.854} C_VEL
LIN {X 0,Y 308.667,Z 893.625,A -85,B 0,C 180,E1 14301.518,E2 14301.518} C_VEL
LIN {X 0,Y 309.41,Z 898.701,A -85,B 0,C 180,E1 14308.595,E2 14308.595} C_VEL
LIN {X 0,Y 308.827,Z 893.926,A -85,B 0,C 180,E1 14317.056,E2 14317.056} C_VEL
LIN {X 0,Y 309.878,Z 874.054,A -85,B 0,C 180,E1 14326.5,E2 14326.5} C_VEL
LIN {X 0,Y 314.949,Z 839.819,A -85,B 0,C 180,E1 14334.746,E2 14334.746} C_VEL
LIN {X 0,Y 322.291,Z 795.815,A -85,B 0,C 180,E1 14340.605,E2 14340.605} C_VEL
LIN {X 0,Y 327.641,Z 744.241,A -85,B 0,C 180,E1 14344.05,E2 14344.05} C_VEL
LIN {X 0,Y 308.874,Z 689.05,A -85,B 0,C 180,E1 14347.268,E2 14347.268} C_VEL
LIN {X 0,Y 299.122,Z 679.829,A -85,B 0,C 180,E1 14349.207,E2 14349.207} C_VEL
LIN {X 0,Y 296.767,Z 678.81,A -85,B 0,C 180,E1 14350.602,E2 14350.602} C_VEL
LIN {X 0,Y 296.793,Z 678.81,A -85,B 0,C 180,E1 14363.978,E2 14363.978} C_VEL
LIN {X 0,Y 297.197,Z 678.81,A -85,B 0,C 180,E1 14374.272,E2 14374.272} C_VEL
LIN {X 0,Y 297.999,Z 678.81,A -85,B 0,C 180,E1 14386.749,E2 14386.749} C_VEL
LIN {X 0,Y 299.196,Z 678.81,A -85,B 0,C 180,E1 14398.544,E2 14398.544} C_VEL
LIN {X 0,Y 298.247,Z 678.81,A -85,B 0,C 180,E1 14413.234,E2 14413.234} C_VEL
LIN {X 0,Y 297.389,Z 678.81,A -85,B 0,C 180,E1 14425.704,E2 14425.704} C_VEL
LIN {X 0,Y 296.763,Z 678.81,A -85,B 0,C 180,E1 14437.569,E2 14437.569} C_VEL
LIN {X 0,Y 296.745,Z 678.81,A -85,B 0,C 180,E1 14450.265,E2 14450.265} C_VEL
LIN {X 0,Y 297.073,Z 678.81,A -85,B 0,C 180,E1 14463.375,E2 14463.375} C_VEL
LIN {X 0,Y 297.983,Z 678.81,A -85,B 0,C 180,E1 14476.752,E2 14476.752} C_VEL
LIN {X 0,Y 298.735,Z 680.834,A -85,B 0,C 180,E1 14482.132,E2 14482.132} C_VEL
LIN {X 0,Y 311.008,Z 720.712,A -85,B 0,C 180,E1 14485.682,E2 14485.682} C_VEL
LIN {X 0,Y 312.689,Z 748.892,A -85,B 0,C 180,E1 14489.113,E2 14489.113} C_VEL
LIN {X 0,Y 306.742,Z 781.944,A -85,B 0,C 180,E1 14495.323,E2 14495.323} C_VEL
LIN {X 0,Y 302.96,Z 802.08,A -85,B 0,C 180,E1 14503.027,E2 14503.027} C_VEL
LIN {X 0,Y 302.242,Z 808.932,A -85,B 0,C 180,E1 14512.122,E2 14512.122} C_VEL
LIN {X 0,Y 305.536,Z 800.858,A -85,B 0,C 180,E1 14520.826,E2 14520.826} C_VEL
LIN {X 0,Y 312.57,Z 778.654,A -85,B 0,C 180,E1 14528.487,E2 14528.487} C_VEL
LIN {X 0,Y 320.465,Z 744.729,A -85,B 0,C 180,E1 14534.247,E2 14534.247} C_VEL
LIN {X 0,Y 310.514,Z 706.84,A -85,B 0,C 180,E1 14539.796,E2 14539.796} C_VEL
LIN {X 0,Y 296.946,Z 678.81,A -85,B 0,C 180,E1 14544.007,E2 14544.007} C_VEL
LIN {X 0,Y 297.189,Z 678.81,A -85,B 0,C 180,E1 14554.278,E2 14554.278} C_VEL
LIN {X 0,Y 297.992,Z 678.81,A -85,B 0,C 180,E1 14566.754,E2 14566.754} C_VEL
LIN {X 0,Y 299.304,Z 678.81,A -85,B 0,C 180,E1 14578.55,E2 14578.55} C_VEL
LIN {X 0,Y 298.433,Z 678.81,A -85,B 0,C 180,E1 14590.256,E2 14590.256} C_VEL
LIN {X 0,Y 297.614,Z 678.81,A -85,B 0,C 180,E1 14602.489,E2 14602.489} C_VEL
LIN {X 0,Y 297.075,Z 678.81,A -85,B 0,C 180,E1 14612.556,E2 14612.556} C_VEL
LIN {X 0,Y 296.893,Z 678.81,A -85,B 0,C 180,E1 14626.021,E2 14626.021} C_VEL
LIN {X 0,Y 323.94,Z 734.585,A -85,B 0,C 180,E1 14632.255,E2 14632.255} C_VEL
LIN {X 0,Y 326.966,Z 754.861,A -85,B 0,C 180,E1 14633.767,E2 14633.767} C_VEL
LIN {X 0,Y 317.966,Z 804.614,A -85,B 0,C 180,E1 14637.728,E2 14637.728} C_VEL
LIN {X 0,Y 307.906,Z 847.145,A -85,B 0,C 180,E1 14644.453,E2 14644.453} C_VEL
LIN {X 0,Y 301.691,Z 878.243,A -85,B 0,C 180,E1 14653.489,E2 14653.489} C_VEL
LIN {X 0,Y 300.78,Z 894.165,A -85,B 0,C 180,E1 14662.754,E2 14662.754} C_VEL
LIN {X 0,Y 301.335,Z 897.208,A -85,B 0,C 180,E1 14671.443,E2 14671.443} C_VEL
LIN {X 0,Y 300.764,Z 887.067,A -85,B 0,C 180,E1 14680.832,E2 14680.832} C_VEL
LIN {X 0,Y 303.05,Z 861.739,A -85,B 0,C 180,E1 14690.137,E2 14690.137} C_VEL
LIN {X 0,Y 309.915,Z 823.461,A -85,B 0,C 180,E1 14697.722,E2 14697.722} C_VEL
LIN {X 0,Y 317.783,Z 775.753,A -85,B 0,C 180,E1 14702.8,E2 14702.8} C_VEL
LIN {X 0,Y 319.145,Z 741.014,A -85,B 0,C 180,E1 14704.881,E2 14704.881} C_VEL
LIN {X 0,Y 296.895,Z 678.81,A -85,B 0,C 180,E1 14708.902,E2 14708.902} C_VEL
LIN {X 0,Y 296.767,Z 678.81,A -85,B 0,C 180,E1 14710.602,E2 14710.602} C_VEL
LIN {X 0,Y 288.562,Z 678.81,A -85,B 0,C 180,E1 14717.409,E2 14717.409} C_VEL
LIN {X 0,Y 288.995,Z 678.81,A -85,B 0,C 180,E1 14730.07,E2 14730.07} C_VEL
LIN {X 0,Y 289.672,Z 678.81,A -85,B 0,C 180,E1 14743.249,E2 14743.249} C_VEL
LIN {X 0,Y 290.757,Z 678.81,A -85,B 0,C 180,E1 14755.506,E2 14755.506} C_VEL
LIN {X 0,Y 290.232,Z 678.81,A -85,B 0,C 180,E1 14767.508,E2 14767.508} C_VEL
LIN {X 0,Y 289.763,Z 678.81,A -85,B 0,C 180,E1 14779.9,E2 14779.9} C_VEL
LIN {X 0,Y 288.871,Z 678.81,A -85,B 0,C 180,E1 14793.476,E2 14793.476} C_VEL
LIN {X 0,Y 288.641,Z 678.81,A -85,B 0,C 180,E1 14805.215,E2 14805.215} C_VEL
LIN {X 0,Y 288.784,Z 678.81,A -85,B 0,C 180,E1 14816.512,E2 14816.512} C_VEL
LIN {X 0,Y 289.189,Z 678.81,A -85,B 0,C 180,E1 14826.823,E2 14826.823} C_VEL
LIN {X 0,Y 290.239,Z 678.81,A -85,B 0,C 180,E1 14839.455,E2 14839.455} C_VEL
LIN {X 0,Y 290.597,Z 680.454,A -85,B 0,C 180,E1 14841.267,E2 14841.267} C_VEL
LIN {X 0,Y 303.482,Z 720.787,A -85,B 0,C 180,E1 14844.981,E2 14844.981} C_VEL
LIN {X 0,Y 305.072,Z 751.127,A -85,B 0,C 180,E1 14848.79,E2 14848.79} C_VEL
LIN {X 0,Y 298.866,Z 783.979,A -85,B 0,C 180,E1 14855.256,E2 14855.256} C_VEL
LIN {X 0,Y 294.917,Z 803.975,A -85,B 0,C 180,E1 14863.389,E2 14863.389} C_VEL
LIN {X 0,Y 294.466,Z 810.058,A -85,B 0,C 180,E1 14872.738,E2 14872.738} C_VEL
LIN {X 0,Y 298.279,Z 801.174,A -85,B 0,C 180,E1 14881.719,E2 14881.719} C_VEL
LIN {X 0,Y 306.087,Z 777.67,A -85,B 0,C 180,E1 14889.617,E2 14889.617} C_VEL
LIN {X 0,Y 313.214,Z 744.004,A -85,B 0,C 180,E1 14895.37,E2 14895.37} C_VEL
LIN {X 0,Y 302.465,Z 705.914,A -85,B 0,C 180,E1 14901.227,E2 14901.227} C_VEL
LIN {X 0,Y 288.81,Z 678.81,A -85,B 0,C 180,E1 14905.571,E2 14905.571} C_VEL
LIN {X 0,Y 289.237,Z 678.81,A -85,B 0,C 180,E1 14916.829,E2 14916.829} C_VEL
LIN {X 0,Y 290.24,Z 678.81,A -85,B 0,C 180,E1 14929.458,E2 14929.458} C_VEL
LIN {X 0,Y 290.993,Z 678.81,A -85,B 0,C 180,E1 14941.497,E2 14941.497} C_VEL
LIN {X 0,Y 290.026,Z 678.81,A -85,B 0,C 180,E1 14954.533,E2 14954.533} C_VEL
LIN {X 0,Y 289.343,Z 678.81,A -85,B 0,C 180,E1 14966.48,E2 14966.48} C_VEL
LIN {X 0,Y 288.877,Z 678.81,A -85,B 0,C 180,E1 14980.383,E2 14980.383} C_VEL
LIN {X 0,Y 288.903,Z 680.002,A -85,B 0,C 180,E1 14984.563,E2 14984.563} C_VEL
LIN {X 0,Y 315.628,Z 731.857,A -85,B 0,C 180,E1 14990.976,E2 14990.976} C_VEL
LIN {X 0,Y 320.347,Z 755.505,A -85,B 0,C 180,E1 14992.986,E2 14992.986} C_VEL
LIN {X 0,Y 310.801,Z 805.218,A -85,B 0,C 180,E1 14997.098,E2 14997.098} C_VEL
LIN {X 0,Y 300.53,Z 846.243,A -85,B 0,C 180,E1 15003.779,E2 15003.779} C_VEL
LIN {X 0,Y 294.006,Z 876.489,A -85,B 0,C 180,E1 15012.747,E2 15012.747} C_VEL
LIN {X 0,Y 292.832,Z 893.047,A -85,B 0,C 180,E1 15022.556,E2 15022.556} C_VEL
LIN {X 0,Y 293.421,Z 895.996,A -85,B 0,C 180,E1 15031.482,E2 15031.482} C_VEL
LIN {X 0,Y 292.822,Z 886.828,A -85,B 0,C 180,E1 15040.45,E2 15040.45} C_VEL
LIN {X 0,Y 294.908,Z 862.709,A -85,B 0,C 180,E1 15049.932,E2 15049.932} C_VEL
LIN {X 0,Y 301.759,Z 825.95,A -85,B 0,C 180,E1 15057.722,E2 15057.722} C_VEL
LIN {X 0,Y 309.944,Z 778.781,A -85,B 0,C 180,E1 15063.109,E2 15063.109} C_VEL
LIN {X 0,Y 311.959,Z 743.331,A -85,B 0,C 180,E1 15065.378,E2 15065.378} C_VEL
LIN {X 0,Y 288.868,Z 678.81,A -85,B 0,C 180,E1 15069.736,E2 15069.736} C_VEL
LIN {X 0,Y 288.562,Z 678.81,A -85,B 0,C 180,E1 15077.409,E2 15077.409} C_VEL
LIN {X 0,Y 280.616,Z 678.81,A -85,B 0,C 180,E1 15084.414,E2 15084.414} C_VEL
LIN {X 0,Y 281.167,Z 678.81,A -85,B 0,C 180,E1 15096.117,E2 15096.117} C_VEL
LIN {X 0,Y 282.16,Z 678.81,A -85,B 0,C 180,E1 15109.146,E2 15109.146} C_VEL
LIN {X 0,Y 283.184,Z 678.81,A -85,B 0,C 180,E1 15118.461,E2 15118.461} C_VEL
LIN {X 0,Y 282.259,Z 678.81,A -85,B 0,C 180,E1 15130.844,E2 15130.844} C_VEL
LIN {X 0,Y 281.409,Z 678.81,A -85,B 0,C 180,E1 15143.855,E2 15143.855} C_VEL
LIN {X 0,Y 280.784,Z 678.81,A -85,B 0,C 180,E1 15154.574,E2 15154.574} C_VEL
LIN {X 0,Y 280.516,Z 678.81,A -85,B 0,C 180,E1 15167.451,E2 15167.451} C_VEL
LIN {X 0,Y 280.78,Z 678.81,A -85,B 0,C 180,E1 15179.106,E2 15179.106} C_VEL
LIN {X 0,Y 281.539,Z 678.81,A -85,B 0,C 180,E1 15192.755,E2 15192.755} C_VEL
LIN {X 0,Y 282.357,Z 679.555,A -85,B 0,C 180,E1 15200.317,E2 15200.317} C_VEL
LIN {X 0,Y 296.175,Z 722.503,A -85,B 0,C 180,E1 15204.422,E2 15204.422} C_VEL
LIN {X 0,Y 297.531,Z 752.711,A -85,B 0,C 180,E1 15208.356,E2 15208.356} C_VEL
LIN {X 0,Y 291.085,Z 785.425,A -85,B 0,C 180,E1 15215.022,E2 15215.022} C_VEL
LIN {X 0,Y 286.903,Z 805.779,A -85,B 0,C 180,E1 15223.77,E2 15223.77} C_VEL
LIN {X 0,Y 286.681,Z 811.134,A -85,B 0,C 180,E1 15233.392,E2 15233.392} C_VEL
LIN {X 0,Y 290.833,Z 802.088,A -85,B 0,C 180,E1 15242.332,E2 15242.332} C_VEL
LIN {X 0,Y 298.932,Z 779.147,A -85,B 0,C 180,E1 15250.223,E2 15250.223} C_VEL
LIN {X 0,Y 306.304,Z 745.546,A -85,B 0,C 180,E1 15256.169,E2 15256.169} C_VEL
LIN {X 0,Y 295.984,Z 708.525,A -85,B 0,C 180,E1 15262.194,E2 15262.194} C_VEL
LIN {X 0,Y 280.777,Z 678.81,A -85,B 0,C 180,E1 15267.533,E2 15267.533} C_VEL
LIN {X 0,Y 281.409,Z 678.81,A -85,B 0,C 180,E1 15280.686,E2 15280.686} C_VEL
LIN {X 0,Y 282.506,Z 678.81,A -85,B 0,C 180,E1 15293.601,E2 15293.601} C_VEL
LIN {X 0,Y 282.776,Z 678.81,A -85,B 0,C 180,E1 15304.621,E2 15304.621} C_VEL
LIN {X 0,Y 281.818,Z 678.81,A -85,B 0,C 180,E1 15317.232,E2 15317.232} C_VEL
LIN {X 0,Y 280.996,Z 678.81,A -85,B 0,C 180,E1 15330.873,E2 15330.873} C_VEL
LIN {X 0,Y 281.051,Z 680.664,A -85,B 0,C 180,E1 15342.867,E2 15342.867} C_VEL
LIN {X 0,Y 307.463,Z 729.591,A -85,B 0,C 180,E1 15349.644,E2 15349.644} C_VEL
LIN {X 0,Y 313.763,Z 756.316,A -85,B 0,C 180,E1 15352.175,E2 15352.175} C_VEL
LIN {X 0,Y 303.688,Z 805.925,A -85,B 0,C 180,E1 15356.441,E2 15356.441} C_VEL
LIN {X 0,Y 292.767,Z 847.004,A -85,B 0,C 180,E1 15363.444,E2 15363.444} C_VEL
LIN {X 0,Y 285.839,Z 877.272,A -85,B 0,C 180,E1 15373.022,E2 15373.022} C_VEL
LIN {X 0,Y 284.863,Z 891.926,A -85,B 0,C 180,E1 15382.346,E2 15382.346} C_VEL
LIN {X 0,Y 285.493,Z 894.78,A -85,B 0,C 180,E1 15391.523,E2 15391.523} C_VEL
LIN {X 0,Y 284.845,Z 885.431,A -85,B 0,C 180,E1 15400.747,E2 15400.747} C_VEL
LIN {X 0,Y 287.174,Z 860.994,A -85,B 0,C 180,E1 15410.493,E2 15410.493} C_VEL
LIN {X 0,Y 294.467,Z 823.579,A -85,B 0,C 180,E1 15418.47,E2 15418.47} C_VEL
LIN {X 0,Y 302.894,Z 776.244,A -85,B 0,C 180,E1 15423.869,E2 15423.869} C_VEL
LIN {X 0,Y 304.467,Z 744.332,A -85,B 0,C 180,E1 15425.992,E2 15425.992} C_VEL
LIN {X 0,Y 280.775,Z 678.81,A -85,B 0,C 180,E1 15430.956,E2 15430.956} C_VEL
LIN {X 0,Y 280.616,Z 678.81,A -85,B 0,C 180,E1 15444.414,E2 15444.414} C_VEL
LIN {X 0,Y 272.873,Z 678.81,A -85,B 0,C 180,E1 15451.631,E2 15451.631} C_VEL
LIN {X 0,Y 273.846,Z 678.81,A -85,B 0,C 180,E1 15465.878,E2 15465.878} C_VEL
LIN {X 0,Y 275.16,Z 678.81,A -85,B 0,C 180,E1 15478.417,E2 15478.417} C_VEL
LIN {X 0,Y 274.206,Z 678.81,A -85,B 0,C 180,E1 15491.166,E2 15491.166} C_VEL
LIN {X 0,Y 273.295,Z 678.81,A -85,B 0,C 180,E1 15504.609,E2 15504.609} C_VEL
LIN {X 0,Y 272.585,Z 678.81,A -85,B 0,C 180,E1 15516.172,E2 15516.172} C_VEL
LIN {X 0,Y 272.429,Z 678.81,A -85,B 0,C 180,E1 15530.164,E2 15530.164} C_VEL
LIN {X 0,Y 272.814,Z 678.81,A -85,B 0,C 180,E1 15541.783,E2 15541.783} C_VEL
LIN {X 0,Y 273.825,Z 678.81,A -85,B 0,C 180,E1 15555.895,E2 15555.895} C_VEL
LIN {X 0,Y 274.357,Z 680.435,A -85,B 0,C 180,E1 15559.387,E2 15559.387} C_VEL
LIN {X 0,Y 288.764,Z 723.188,A -85,B 0,C 180,E1 15563.733,E2 15563.733} C_VEL
LIN {X 0,Y 290.015,Z 754.34,A -85,B 0,C 180,E1 15567.912,E2 15567.912} C_VEL
LIN {X 0,Y 283.416,Z 786.281,A -85,B 0,C 180,E1 15574.607,E2 15574.607} C_VEL
LIN {X 0,Y 279.069,Z 806.572,A -85,B 0,C 180,E1 15583.418,E2 15583.418} C_VEL
LIN {X 0,Y 278.338,Z 812.346,A -85,B 0,C 180,E1 15590.756,E2 15590.756} C_VEL
LIN {X 0,Y 281.79,Z 806.623,A -85,B 0,C 180,E1 15600.771,E2 15600.771} C_VEL
LIN {X 0,Y 289.786,Z 786.178,A -85,B 0,C 180,E1 15609.418,E2 15609.418} C_VEL
LIN {X 0,Y 299.84,Z 752.268,A -85,B 0,C 180,E1 15616.072,E2 15616.072} C_VEL
LIN {X 0,Y 291.674,Z 716.4,A -85,B 0,C 180,E1 15622.315,E2 15622.315} C_VEL
LIN {X 0,Y 272.858,Z 678.81,A -85,B 0,C 180,E1 15628.982,E2 15628.982} C_VEL
LIN {X 0,Y 273.523,Z 678.81,A -85,B 0,C 180,E1 15642.235,E2 15642.235} C_VEL
LIN {X 0,Y 274.708,Z 678.81,A -85,B 0,C 180,E1 15655.25,E2 15655.25} C_VEL
LIN {X 0,Y 274.593,Z 678.81,A -85,B 0,C 180,E1 15667.945,E2 15667.945} C_VEL
LIN {X 0,Y 273.491,Z 678.81,A -85,B 0,C 180,E1 15681.146,E2 15681.146} C_VEL
LIN {X 0,Y 272.925,Z 678.81,A -85,B 0,C 180,E1 15691.892,E2 15691.892} C_VEL
LIN {X 0,Y 272.847,Z 680.664,A -85,B 0,C 180,E1 15700.882,E2 15700.882} C_VEL
LIN {X 0,Y 299.469,Z 727.915,A -85,B 0,C 180,E1 15708.242,E2 15708.242} C_VEL
LIN {X 0,Y 307.268,Z 757.061,A -85,B 0,C 180,E1 15711.328,E2 15711.328} C_VEL
LIN {X 0,Y 296.949,Z 805.239,A -85,B 0,C 180,E1 15715.574,E2 15715.574} C_VEL
LIN {X 0,Y 285.464,Z 846.13,A -85,B 0,C 180,E1 15722.709,E2 15722.709} C_VEL
LIN {X 0,Y 278.044,Z 876.255,A -85,B 0,C 180,E1 15732.531,E2 15732.531} C_VEL
LIN {X 0,Y 277.066,Z 892.097,A -85,B 0,C 180,E1 15743.711,E2 15743.711} C_VEL
LIN {X 0,Y 277.577,Z 893.565,A -85,B 0,C 180,E1 15751.566,E2 15751.566} C_VEL
LIN {X 0,Y 276.878,Z 884.026,A -85,B 0,C 180,E1 15761.06,E2 15761.06} C_VEL
LIN {X 0,Y 279.235,Z 860.524,A -85,B 0,C 180,E1 15770.686,E2 15770.686} C_VEL
LIN {X 0,Y 286.888,Z 822.971,A -85,B 0,C 180,E1 15778.973,E2 15778.973} C_VEL
LIN {X 0,Y 295.517,Z 776.275,A -85,B 0,C 180,E1 15784.462,E2 15784.462} C_VEL
LIN {X 0,Y 297.157,Z 745.821,A -85,B 0,C 180,E1 15786.594,E2 15786.594} C_VEL
LIN {X 0,Y 272.677,Z 678.81,A -85,B 0,C 180,E1 15791.671,E2 15791.671} C_VEL
LIN {X 0,Y 272.582,Z 678.81,A -85,B 0,C 180,E1 15804.383,E2 15804.383} C_VEL
LIN {X 0,Y 272.873,Z 678.81,A -85,B 0,C 180,E1 15811.631,E2 15811.631} C_VEL
LIN {X 0,Y 265.138,Z 678.81,A -85,B 0,C 180,E1 15819.016,E2 15819.016} C_VEL
LIN {X 0,Y 266.369,Z 678.81,A -85,B 0,C 180,E1 15831.808,E2 15831.808} C_VEL
LIN {X 0,Y 266.315,Z 678.81,A -85,B 0,C 180,E1 15841.629,E2 15841.629} C_VEL
LIN {X 0,Y 265.983,Z 678.81,A -85,B 0,C 180,E1 15854.874,E2 15854.874} C_VEL
LIN {X 0,Y 265.012,Z 678.81,A -85,B 0,C 180,E1 15867.429,E2 15867.429} C_VEL
LIN {X 0,Y 264.44,Z 678.81,A -85,B 0,C 180,E1 15881.294,E2 15881.294} C_VEL
LIN {X 0,Y 264.423,Z 678.81,A -85,B 0,C 180,E1 15892.944,E2 15892.944} C_VEL
LIN {X 0,Y 264.882,Z 678.81,A -85,B 0,C 180,E1 15904.553,E2 15904.553} C_VEL
LIN {X 0,Y 266.243,Z 680.721,A -85,B 0,C 180,E1 15918.379,E2 15918.379} C_VEL
LIN {X 0,Y 281.21,Z 722.463,A -85,B 0,C 180,E1 15922.844,E2 15922.844} C_VEL
LIN {X 0,Y 282.628,Z 755.01,A -85,B 0,C 180,E1 15927.307,E2 15927.307} C_VEL
LIN {X 0,Y 275.641,Z 787.665,A -85,B 0,C 180,E1 15934.342,E2 15934.342} C_VEL
LIN {X 0,Y 271.198,Z 807.523,A -85,B 0,C 180,E1 15943.191,E2 15943.191} C_VEL
LIN {X 0,Y 270.632,Z 813.679,A -85,B 0,C 180,E1 15952.299,E2 15952.299} C_VEL
LIN {X 0,Y 274.508,Z 807.214,A -85,B 0,C 180,E1 15961.681,E2 15961.681} C_VEL
LIN {X 0,Y 283.235,Z 785.972,A -85,B 0,C 180,E1 15970.515,E2 15970.515} C_VEL
LIN {X 0,Y 292.901,Z 752.502,A -85,B 0,C 180,E1 15977.18,E2 15977.18} C_VEL
LIN {X 0,Y 284.317,Z 716.296,A -85,B 0,C 180,E1 15983.812,E2 15983.812} C_VEL
LIN {X 0,Y 264.838,Z 678.81,A -85,B 0,C 180,E1 15991.34,E2 15991.34} C_VEL
LIN {X 0,Y 265.677,Z 678.81,A -85,B 0,C 180,E1 16005.108,E2 16005.108} C_VEL
LIN {X 0,Y 267.219,Z 678.81,A -85,B 0,C 180,E1 16018.376,E2 16018.376} C_VEL
LIN {X 0,Y 266.21,Z 678.81,A -85,B 0,C 180,E1 16031.513,E2 16031.513} C_VEL
LIN {X 0,Y 265.149,Z 678.81,A -85,B 0,C 180,E1 16045.425,E2 16045.425} C_VEL
LIN {X 0,Y 264.82,Z 680.82,A -85,B 0,C 180,E1 16058.701,E2 16058.701} C_VEL
LIN {X 0,Y 290.82,Z 724.8,A -85,B 0,C 180,E1 16066.531,E2 16066.531} C_VEL
LIN {X 0,Y 300.838,Z 757.87,A -85,B 0,C 180,E1 16070.443,E2 16070.443} C_VEL
LIN {X 0,Y 289.917,Z 805.966,A -85,B 0,C 180,E1 16074.845,E2 16074.845} C_VEL
LIN {X 0,Y 277.706,Z 846.841,A -85,B 0,C 180,E1 16082.323,E2 16082.323} C_VEL
LIN {X 0,Y 269.947,Z 876.614,A -85,B 0,C 180,E1 16092.689,E2 16092.689} C_VEL
LIN {X 0,Y 269.115,Z 890.973,A -85,B 0,C 180,E1 16103.524,E2 16103.524} C_VEL
LIN {X 0,Y 269.645,Z 892.343,A -85,B 0,C 180,E1 16111.612,E2 16111.612} C_VEL
LIN {X 0,Y 268.913,Z 882.577,A -85,B 0,C 180,E1 16121.392,E2 16121.392} C_VEL
LIN {X 0,Y 271.521,Z 858.761,A -85,B 0,C 180,E1 16131.302,E2 16131.302} C_VEL
LIN {X 0,Y 279.56,Z 821.018,A -85,B 0,C 180,E1 16139.722,E2 16139.722} C_VEL
LIN {X 0,Y 288.351,Z 775.112,A -85,B 0,C 180,E1 16145.174,E2 16145.174} C_VEL
LIN {X 0,Y 289.762,Z 747.298,A -85,B 0,C 180,E1 16147.201,E2 16147.201} C_VEL
LIN {X 0,Y 266.18,Z 683.547,A -85,B 0,C 180,E1 16152.199,E2 16152.199} C_VEL
LIN {X 0,Y 264.587,Z 678.81,A -85,B 0,C 180,E1 16152.804,E2 16152.804} C_VEL
LIN {X 0,Y 264.623,Z 678.81,A -85,B 0,C 180,E1 16166.983,E2 16166.983} C_VEL
LIN {X 0,Y 265.138,Z 678.81,A -85,B 0,C 180,E1 16179.016,E2 16179.016} C_VEL
LIN {X 0,Y 257.732,Z 678.81,A -85,B 0,C 180,E1 16186.639,E2 16186.639} C_VEL
LIN {X 0,Y 259.131,Z 678.81,A -85,B 0,C 180,E1 16198.319,E2 16198.319} C_VEL
LIN {X 0,Y 257.954,Z 678.81,A -85,B 0,C 180,E1 16213.905,E2 16213.905} C_VEL
LIN {X 0,Y 257.042,Z 678.81,A -85,B 0,C 180,E1 16226.28,E2 16226.28} C_VEL
LIN {X 0,Y 256.405,Z 678.81,A -85,B 0,C 180,E1 16238.42,E2 16238.42} C_VEL
LIN {X 0,Y 256.424,Z 678.81,A -85,B 0,C 180,E1 16253.028,E2 16253.028} C_VEL
LIN {X 0,Y 256.974,Z 678.81,A -85,B 0,C 180,E1 16267.428,E2 16267.428} C_VEL
LIN {X 0,Y 257.893,Z 679.32,A -85,B 0,C 180,E1 16277.204,E2 16277.204} C_VEL
LIN {X 0,Y 273.658,Z 723,A -85,B 0,C 180,E1 16282.031,E2 16282.031} C_VEL
LIN {X 0,Y 275.124,Z 756.713,A -85,B 0,C 180,E1 16286.838,E2 16286.838} C_VEL
LIN {X 0,Y 267.876,Z 789.034,A -85,B 0,C 180,E1 16294.061,E2 16294.061} C_VEL
LIN {X 0,Y 263.233,Z 808.965,A -85,B 0,C 180,E1 16303.333,E2 16303.333} C_VEL
LIN {X 0,Y 262.694,Z 814.865,A -85,B 0,C 180,E1 16312.055,E2 16312.055} C_VEL
LIN {X 0,Y 266.462,Z 809.279,A -85,B 0,C 180,E1 16321.526,E2 16321.526} C_VEL
LIN {X 0,Y 275.42,Z 789.112,A -85,B 0,C 180,E1 16330.71,E2 16330.71} C_VEL
LIN {X 0,Y 286.208,Z 756.272,A -85,B 0,C 180,E1 16337.641,E2 16337.641} C_VEL
LIN {X 0,Y 279.272,Z 722.257,A -85,B 0,C 180,E1 16344.259,E2 16344.259} C_VEL
LIN {X 0,Y 260.12,Z 685.216,A -85,B 0,C 180,E1 16352.224,E2 16352.224} C_VEL
LIN {X 0,Y 256.868,Z 678.81,A -85,B 0,C 180,E1 16353.701,E2 16353.701} C_VEL
LIN {X 0,Y 257.951,Z 678.81,A -85,B 0,C 180,E1 16368.12,E2 16368.12} C_VEL
LIN {X 0,Y 259.208,Z 678.81,A -85,B 0,C 180,E1 16378.326,E2 16378.326} C_VEL
LIN {X 0,Y 258.127,Z 678.81,A -85,B 0,C 180,E1 16391.879,E2 16391.879} C_VEL
LIN {X 0,Y 257.139,Z 678.81,A -85,B 0,C 180,E1 16403.829,E2 16403.829} C_VEL
LIN {X 0,Y 256.683,Z 680.156,A -85,B 0,C 180,E1 16416.166,E2 16416.166} C_VEL
LIN {X 0,Y 282.641,Z 723.168,A -85,B 0,C 180,E1 16424.813,E2 16424.813} C_VEL
LIN {X 0,Y 294.441,Z 758.992,A -85,B 0,C 180,E1 16429.528,E2 16429.528} C_VEL
LIN {X 0,Y 282.712,Z 807.373,A -85,B 0,C 180,E1 16434.188,E2 16434.188} C_VEL
LIN {X 0,Y 269.975,Z 847.512,A -85,B 0,C 180,E1 16441.916,E2 16441.916} C_VEL
LIN {X 0,Y 262.048,Z 876.118,A -85,B 0,C 180,E1 16452.414,E2 16452.414} C_VEL
LIN {X 0,Y 261.135,Z 889.843,A -85,B 0,C 180,E1 16463.325,E2 16463.325} C_VEL
LIN {X 0,Y 261.726,Z 891.122,A -85,B 0,C 180,E1 16471.661,E2 16471.661} C_VEL
LIN {X 0,Y 260.963,Z 881.109,A -85,B 0,C 180,E1 16481.743,E2 16481.743} C_VEL
LIN {X 0,Y 263.894,Z 856.968,A -85,B 0,C 180,E1 16491.949,E2 16491.949} C_VEL
LIN {X 0,Y 272.371,Z 818.794,A -85,B 0,C 180,E1 16500.539,E2 16500.539} C_VEL
LIN {X 0,Y 281.621,Z 771.56,A -85,B 0,C 180,E1 16506.107,E2 16506.107} C_VEL
LIN {X 0,Y 282.35,Z 748.514,A -85,B 0,C 180,E1 16507.86,E2 16507.86} C_VEL
LIN {X 0,Y 260.304,Z 688.139,A -85,B 0,C 180,E1 16512.845,E2 16512.845} C_VEL
LIN {X 0,Y 256.468,Z 678.81,A -85,B 0,C 180,E1 16514.07,E2 16514.07} C_VEL
LIN {X 0,Y 256.52,Z 678.81,A -85,B 0,C 180,E1 16525.799,E2 16525.799} C_VEL
LIN {X 0,Y 257.032,Z 678.81,A -85,B 0,C 180,E1 16539.04,E2 16539.04} C_VEL
LIN {X 0,Y 257.732,Z 678.81,A -85,B 0,C 180,E1 16546.639,E2 16546.639} C_VEL
LIN {X 0,Y 250.574,Z 678.81,A -85,B 0,C 180,E1 16554.523,E2 16554.523} C_VEL
LIN {X 0,Y 250.064,Z 678.81,A -85,B 0,C 180,E1 16565.22,E2 16565.22} C_VEL
LIN {X 0,Y 249.783,Z 678.81,A -85,B 0,C 180,E1 16575.864,E2 16575.864} C_VEL
LIN {X 0,Y 248.793,Z 678.81,A -85,B 0,C 180,E1 16587.817,E2 16587.817} C_VEL
LIN {X 0,Y 248.241,Z 678.81,A -85,B 0,C 180,E1 16600.169,E2 16600.169} C_VEL
LIN {X 0,Y 248.446,Z 678.81,A -85,B 0,C 180,E1 16615.546,E2 16615.546} C_VEL
LIN {X 0,Y 249.148,Z 678.81,A -85,B 0,C 180,E1 16630.428,E2 16630.428} C_VEL
LIN {X 0,Y 249.825,Z 680.08,A -85,B 0,C 180,E1 16636.055,E2 16636.055} C_VEL
LIN {X 0,Y 265.82,Z 722.432,A -85,B 0,C 180,E1 16641.026,E2 16641.026} C_VEL
LIN {X 0,Y 267.839,Z 757.128,A -85,B 0,C 180,E1 16646.126,E2 16646.126} C_VEL
LIN {X 0,Y 260.375,Z 789.12,A -85,B 0,C 180,E1 16653.341,E2 16653.341} C_VEL
LIN {X 0,Y 255.448,Z 809.635,A -85,B 0,C 180,E1 16662.872,E2 16662.872} C_VEL
LIN {X 0,Y 254.896,Z 816.046,A -85,B 0,C 180,E1 16672.767,E2 16672.767} C_VEL
LIN {X 0,Y 259.283,Z 809.847,A -85,B 0,C 180,E1 16682.559,E2 16682.559} C_VEL
LIN {X 0,Y 268.88,Z 789.35,A -85,B 0,C 180,E1 16691.789,E2 16691.789} C_VEL
LIN {X 0,Y 279.417,Z 757.004,A -85,B 0,C 180,E1 16698.756,E2 16698.756} C_VEL
LIN {X 0,Y 272.078,Z 722.215,A -85,B 0,C 180,E1 16705.918,E2 16705.918} C_VEL
LIN {X 0,Y 252.898,Z 685.778,A -85,B 0,C 180,E1 16714.577,E2 16714.577} C_VEL
LIN {X 0,Y 248.942,Z 678.81,A -85,B 0,C 180,E1 16716.659,E2 16716.659} C_VEL
LIN {X 0,Y 250.243,Z 678.81,A -85,B 0,C 180,E1 16731.283,E2 16731.283} C_VEL
LIN {X 0,Y 250.764,Z 678.81,A -85,B 0,C 180,E1 16743.104,E2 16743.104} C_VEL
LIN {X 0,Y 249.73,Z 678.81,A -85,B 0,C 180,E1 16755.874,E2 16755.874} C_VEL
LIN {X 0,Y 248.826,Z 678.81,A -85,B 0,C 180,E1 16767.831,E2 16767.831} C_VEL
LIN {X 0,Y 248.877,Z 680.881,A -85,B 0,C 180,E1 16773.421,E2 16773.421} C_VEL
LIN {X 0,Y 273.371,Z 719.539,A -85,B 0,C 180,E1 16782.582,E2 16782.582} C_VEL
LIN {X 0,Y 287.94,Z 759.047,A -85,B 0,C 180,E1 16788.454,E2 16788.454} C_VEL
LIN {X 0,Y 275.908,Z 807.683,A -85,B 0,C 180,E1 16793.334,E2 16793.334} C_VEL
LIN {X 0,Y 262.783,Z 846.664,A -85,B 0,C 180,E1 16801.076,E2 16801.076} C_VEL
LIN {X 0,Y 254.312,Z 874.826,A -85,B 0,C 180,E1 16811.695,E2 16811.695} C_VEL
LIN {X 0,Y 253.035,Z 887.812,A -85,B 0,C 180,E1 16821.762,E2 16821.762} C_VEL
LIN {X 0,Y 253.79,Z 889.898,A -85,B 0,C 180,E1 16831.713,E2 16831.713} C_VEL
LIN {X 0,Y 253.031,Z 879.64,A -85,B 0,C 180,E1 16842.117,E2 16842.117} C_VEL
LIN {X 0,Y 256.304,Z 855.104,A -85,B 0,C 180,E1 16852.635,E2 16852.635} C_VEL
LIN {X 0,Y 265.154,Z 816.738,A -85,B 0,C 180,E1 16861.37,E2 16861.37} C_VEL
LIN {X 0,Y 274.851,Z 768.708,A -85,B 0,C 180,E1 16867.025,E2 16867.025} C_VEL
LIN {X 0,Y 274.513,Z 747.775,A -85,B 0,C 180,E1 16868.735,E2 16868.735} C_VEL
LIN {X 0,Y 252.418,Z 688.378,A -85,B 0,C 180,E1 16873.956,E2 16873.956} C_VEL
LIN {X 0,Y 248.354,Z 678.81,A -85,B 0,C 180,E1 16875.348,E2 16875.348} C_VEL
LIN {X 0,Y 248.577,Z 678.81,A -85,B 0,C 180,E1 16888.734,E2 16888.734} C_VEL
LIN {X 0,Y 249.236,Z 678.81,A -85,B 0,C 180,E1 16900.693,E2 16900.693} C_VEL
LIN {X 0,Y 250.574,Z 678.81,A -85,B 0,C 180,E1 16914.523,E2 16914.523} C_VEL
LIN {X 0,Y 242.143,Z 678.81,A -85,B 0,C 180,E1 16922.605,E2 16922.605} C_VEL
LIN {X 0,Y 241.698,Z 678.81,A -85,B 0,C 180,E1 16936.409,E2 16936.409} C_VEL
LIN {X 0,Y 240.736,Z 678.81,A -85,B 0,C 180,E1 16948.213,E2 16948.213} C_VEL
LIN {X 0,Y 240.06,Z 678.81,A -85,B 0,C 180,E1 16963.367,E2 16963.367} C_VEL
LIN {X 0,Y 240.474,Z 678.81,A -85,B 0,C 180,E1 16978.421,E2 16978.421} C_VEL
LIN {X 0,Y 241.359,Z 678.81,A -85,B 0,C 180,E1 16993.565,E2 16993.565} C_VEL
LIN {X 0,Y 241.739,Z 680.553,A -85,B 0,C 180,E1 16994.821,E2 16994.821} C_VEL
LIN {X 0,Y 257.947,Z 721.975,A -85,B 0,C 180,E1 16999.977,E2 16999.977} C_VEL
LIN {X 0,Y 260.695,Z 756.98,A -85,B 0,C 180,E1 17005.296,E2 17005.296} C_VEL
LIN {X 0,Y 252.695,Z 790.157,A -85,B 0,C 180,E1 17012.905,E2 17012.905} C_VEL
LIN {X 0,Y 247.643,Z 810.248,A -85,B 0,C 180,E1 17022.385,E2 17022.385} C_VEL
LIN {X 0,Y 247.141,Z 817.231,A -85,B 0,C 180,E1 17033.524,E2 17033.524} C_VEL
LIN {X 0,Y 252.213,Z 810.247,A -85,B 0,C 180,E1 17043.73,E2 17043.73} C_VEL
LIN {X 0,Y 262.651,Z 789.084,A -85,B 0,C 180,E1 17053.058,E2 17053.058} C_VEL
LIN {X 0,Y 272.715,Z 758.369,A -85,B 0,C 180,E1 17059.81,E2 17059.81} C_VEL
LIN {X 0,Y 265.83,Z 724.742,A -85,B 0,C 180,E1 17067.16,E2 17067.16} C_VEL
LIN {X 0,Y 248.501,Z 691.58,A -85,B 0,C 180,E1 17075.837,E2 17075.837} C_VEL
LIN {X 0,Y 241.118,Z 678.81,A -85,B 0,C 180,E1 17079.75,E2 17079.75} C_VEL
LIN {X 0,Y 242.583,Z 678.81,A -85,B 0,C 180,E1 17094.619,E2 17094.619} C_VEL
LIN {X 0,Y 242.677,Z 678.81,A -85,B 0,C 180,E1 17105.386,E2 17105.386} C_VEL
LIN {X 0,Y 241.309,Z 678.81,A -85,B 0,C 180,E1 17120.241,E2 17120.241} C_VEL
LIN {X 0,Y 240.822,Z 680.389,A -85,B 0,C 180,E1 17130.008,E2 17130.008} C_VEL
LIN {X 0,Y 264.537,Z 716.71,A -85,B 0,C 180,E1 17140.2,E2 17140.2} C_VEL
LIN {X 0,Y 280.268,Z 755.49,A -85,B 0,C 180,E1 17146.723,E2 17146.723} C_VEL
LIN {X 0,Y 280.027,Z 769.625,A -85,B 0,C 180,E1 17148.23,E2 17148.23} C_VEL
LIN {X 0,Y 266.694,Z 815.258,A -85,B 0,C 180,E1 17153.564,E2 17153.564} C_VEL
LIN {X 0,Y 253.004,Z 852.946,A -85,B 0,C 180,E1 17162.299,E2 17162.299} C_VEL
LIN {X 0,Y 245.456,Z 878.313,A -85,B 0,C 180,E1 17173.846,E2 17173.846} C_VEL
LIN {X 0,Y 245.408,Z 888.473,A -85,B 0,C 180,E1 17184.678,E2 17184.678} C_VEL
LIN {X 0,Y 245.582,Z 886.608,A -85,B 0,C 180,E1 17195.318,E2 17195.318} C_VEL
LIN {X 0,Y 246.14,Z 869.657,A -85,B 0,C 180,E1 17207.109,E2 17207.109} C_VEL
LIN {X 0,Y 252.304,Z 839.089,A -85,B 0,C 180,E1 17217.298,E2 17217.298} C_VEL
LIN {X 0,Y 262.132,Z 796.706,A -85,B 0,C 180,E1 17224.868,E2 17224.868} C_VEL
LIN {X 0,Y 268.369,Z 754.094,A -85,B 0,C 180,E1 17228.957,E2 17228.957} C_VEL
LIN {X 0,Y 249.911,Z 700.171,A -85,B 0,C 180,E1 17233.944,E2 17233.944} C_VEL
LIN {X 0,Y 240.193,Z 678.81,A -85,B 0,C 180,E1 17236.6,E2 17236.6} C_VEL
LIN {X 0,Y 240.622,Z 678.81,A -85,B 0,C 180,E1 17251.764,E2 17251.764} C_VEL
LIN {X 0,Y 241.685,Z 678.81,A -85,B 0,C 180,E1 17266.717,E2 17266.717} C_VEL
LIN {X 0,Y 243.087,Z 678.81,A -85,B 0,C 180,E1 17278.208,E2 17278.208} C_VEL
LIN {X 0,Y 242.143,Z 678.81,A -85,B 0,C 180,E1 17282.605,E2 17282.605} C_VEL
LIN {X 0,Y 233.837,Z 678.81,A -85,B 0,C 180,E1 17290.936,E2 17290.936} C_VEL
LIN {X 0,Y 232.863,Z 678.81,A -85,B 0,C 180,E1 17305.059,E2 17305.059} C_VEL
LIN {X 0,Y 232.077,Z 678.81,A -85,B 0,C 180,E1 17318.402,E2 17318.402} C_VEL
LIN {X 0,Y 232.048,Z 678.81,A -85,B 0,C 180,E1 17331.59,E2 17331.59} C_VEL
LIN {X 0,Y 232.609,Z 678.81,A -85,B 0,C 180,E1 17344.909,E2 17344.909} C_VEL
LIN {X 0,Y 233.414,Z 680.005,A -85,B 0,C 180,E1 17353.403,E2 17353.403} C_VEL
LIN {X 0,Y 250.429,Z 722.567,A -85,B 0,C 180,E1 17359.01,E2 17359.01} C_VEL
LIN {X 0,Y 253.423,Z 757.663,A -85,B 0,C 180,E1 17364.565,E2 17364.565} C_VEL
LIN {X 0,Y 244.974,Z 791.393,A -85,B 0,C 180,E1 17372.515,E2 17372.515} C_VEL
LIN {X 0,Y 239.573,Z 812.097,A -85,B 0,C 180,E1 17382.809,E2 17382.809} C_VEL
LIN {X 0,Y 239.44,Z 818.403,A -85,B 0,C 180,E1 17394.328,E2 17394.328} C_VEL
LIN {X 0,Y 245.336,Z 810.538,A -85,B 0,C 180,E1 17405.009,E2 17405.009} C_VEL
LIN {X 0,Y 257.041,Z 787.735,A -85,B 0,C 180,E1 17414.699,E2 17414.699} C_VEL
LIN {X 0,Y 266.129,Z 760.815,A -85,B 0,C 180,E1 17420.674,E2 17420.674} C_VEL
LIN {X 0,Y 260.226,Z 728.56,A -85,B 0,C 180,E1 17428.148,E2 17428.148} C_VEL
LIN {X 0,Y 244.339,Z 696.904,A -85,B 0,C 180,E1 17437.077,E2 17437.077} C_VEL
LIN {X 0,Y 233.405,Z 678.81,A -85,B 0,C 180,E1 17443.962,E2 17443.962} C_VEL
LIN {X 0,Y 235.13,Z 678.81,A -85,B 0,C 180,E1 17458.154,E2 17458.154} C_VEL
LIN {X 0,Y 234.257,Z 678.81,A -85,B 0,C 180,E1 17469.325,E2 17469.325} C_VEL
LIN {X 0,Y 233.176,Z 678.81,A -85,B 0,C 180,E1 17480.98,E2 17480.98} C_VEL
LIN {X 0,Y 233.028,Z 680.818,A -85,B 0,C 180,E1 17486.011,E2 17486.011} C_VEL
LIN {X 0,Y 251.816,Z 708.033,A -85,B 0,C 180,E1 17495.912,E2 17495.912} C_VEL
LIN {X 0,Y 270.398,Z 745.239,A -85,B 0,C 180,E1 17503.7,E2 17503.7} C_VEL
LIN {X 0,Y 274.453,Z 767.942,A -85,B 0,C 180,E1 17507.002,E2 17507.002} C_VEL
LIN {X 0,Y 260.229,Z 814.633,A -85,B 0,C 180,E1 17512.506,E2 17512.506} C_VEL
LIN {X 0,Y 245.805,Z 852.12,A -85,B 0,C 180,E1 17521.414,E2 17521.414} C_VEL
LIN {X 0,Y 237.647,Z 877.285,A -85,B 0,C 180,E1 17533.3,E2 17533.3} C_VEL
LIN {X 0,Y 237.44,Z 887.328,A -85,B 0,C 180,E1 17544.499,E2 17544.499} C_VEL
LIN {X 0,Y 237.715,Z 886.533,A -85,B 0,C 180,E1 17553.66,E2 17553.66} C_VEL
LIN {X 0,Y 237.526,Z 873.565,A -85,B 0,C 180,E1 17564.807,E2 17564.807} C_VEL
LIN {X 0,Y 242.652,Z 845.985,A -85,B 0,C 180,E1 17575.763,E2 17575.763} C_VEL
LIN {X 0,Y 252.703,Z 805.698,A -85,B 0,C 180,E1 17584.263,E2 17584.263} C_VEL
LIN {X 0,Y 261.494,Z 757.766,A -85,B 0,C 180,E1 17589.423,E2 17589.423} C_VEL
LIN {X 0,Y 245.104,Z 707.091,A -85,B 0,C 180,E1 17594.434,E2 17594.434} C_VEL
LIN {X 0,Y 232.154,Z 678.81,A -85,B 0,C 180,E1 17597.783,E2 17597.783} C_VEL
LIN {X 0,Y 232.632,Z 678.81,A -85,B 0,C 180,E1 17611.721,E2 17611.721} C_VEL
LIN {X 0,Y 233.709,Z 678.81,A -85,B 0,C 180,E1 17626.859,E2 17626.859} C_VEL
LIN {X 0,Y 235.071,Z 678.81,A -85,B 0,C 180,E1 17638.146,E2 17638.146} C_VEL
LIN {X 0,Y 233.837,Z 678.81,A -85,B 0,C 180,E1 17650.936,E2 17650.936} C_VEL
LIN {X 0,Y 225.123,Z 678.81,A -85,B 0,C 180,E1 17659.558,E2 17659.558} C_VEL
LIN {X 0,Y 224.249,Z 678.81,A -85,B 0,C 180,E1 17672.231,E2 17672.231} C_VEL
LIN {X 0,Y 223.981,Z 678.81,A -85,B 0,C 180,E1 17685.347,E2 17685.347} C_VEL
LIN {X 0,Y 224.24,Z 678.81,A -85,B 0,C 180,E1 17699.499,E2 17699.499} C_VEL
LIN {X 0,Y 225.267,Z 680.374,A -85,B 0,C 180,E1 17711.925,E2 17711.925} C_VEL
LIN {X 0,Y 242.592,Z 721.711,A -85,B 0,C 180,E1 17717.77,E2 17717.77} C_VEL
LIN {X 0,Y 246.887,Z 755.169,A -85,B 0,C 180,E1 17723.262,E2 17723.262} C_VEL
LIN {X 0,Y 238.157,Z 789.089,A -85,B 0,C 180,E1 17730.913,E2 17730.913} C_VEL
LIN {X 0,Y 232.349,Z 810.461,A -85,B 0,C 180,E1 17740.621,E2 17740.621} C_VEL
LIN {X 0,Y 230.905,Z 819.3,A -85,B 0,C 180,E1 17751.191,E2 17751.191} C_VEL
LIN {X 0,Y 235.836,Z 814.889,A -85,B 0,C 180,E1 17763.158,E2 17763.158} C_VEL
LIN {X 0,Y 246.952,Z 795.742,A -85,B 0,C 180,E1 17773.537,E2 17773.537} C_VEL
LIN {X 0,Y 259.582,Z 764.611,A -85,B 0,C 180,E1 17781.248,E2 17781.248} C_VEL
LIN {X 0,Y 254.736,Z 732.964,A -85,B 0,C 180,E1 17789.034,E2 17789.034} C_VEL
LIN {X 0,Y 239.508,Z 699.958,A -85,B 0,C 180,E1 17798.911,E2 17798.911} C_VEL
LIN {X 0,Y 227.252,Z 683.499,A -85,B 0,C 180,E1 17807.278,E2 17807.278} C_VEL
LIN {X 0,Y 225.879,Z 678.81,A -85,B 0,C 180,E1 17809.619,E2 17809.619} C_VEL
LIN {X 0,Y 226.919,Z 678.81,A -85,B 0,C 180,E1 17821.92,E2 17821.92} C_VEL
LIN {X 0,Y 225.782,Z 678.81,A -85,B 0,C 180,E1 17833.611,E2 17833.611} C_VEL
LIN {X 0,Y 225.475,Z 680.852,A -85,B 0,C 180,E1 17840.824,E2 17840.824} C_VEL
LIN {X 0,Y 240.793,Z 702.462,A -85,B 0,C 180,E1 17851.39,E2 17851.39} C_VEL
LIN {X 0,Y 260.025,Z 736.62,A -85,B 0,C 180,E1 17860.357,E2 17860.357} C_VEL
LIN {X 0,Y 268.42,Z 768.684,A -85,B 0,C 180,E1 17865.911,E2 17865.911} C_VEL
LIN {X 0,Y 253.857,Z 814.076,A -85,B 0,C 180,E1 17871.395,E2 17871.395} C_VEL
LIN {X 0,Y 238.621,Z 851.281,A -85,B 0,C 180,E1 17880.47,E2 17880.47} C_VEL
LIN {X 0,Y 229.836,Z 876.271,A -85,B 0,C 180,E1 17892.715,E2 17892.715} C_VEL
LIN {X 0,Y 229.47,Z 886.182,A -85,B 0,C 180,E1 17904.307,E2 17904.307} C_VEL
LIN {X 0,Y 229.789,Z 885.253,A -85,B 0,C 180,E1 17913.786,E2 17913.786} C_VEL
LIN {X 0,Y 229.91,Z 870.629,A -85,B 0,C 180,E1 17926.129,E2 17926.129} C_VEL
LIN {X 0,Y 235.892,Z 841.745,A -85,B 0,C 180,E1 17937.282,E2 17937.282} C_VEL
LIN {X 0,Y 246.242,Z 801.282,A -85,B 0,C 180,E1 17945.564,E2 17945.564} C_VEL
LIN {X 0,Y 253.644,Z 756.625,A -85,B 0,C 180,E1 17950.442,E2 17950.442} C_VEL
LIN {X 0,Y 237.407,Z 707.289,A -85,B 0,C 180,E1 17955.633,E2 17955.633} C_VEL
LIN {X 0,Y 224.086,Z 678.81,A -85,B 0,C 180,E1 17959.208,E2 17959.208} C_VEL
LIN {X 0,Y 224.573,Z 678.81,A -85,B 0,C 180,E1 17973.939,E2 17973.939} C_VEL
LIN {X 0,Y 225.721,Z 678.81,A -85,B 0,C 180,E1 17987.122,E2 17987.122} C_VEL
LIN {X 0,Y 227.036,Z 678.81,A -85,B 0,C 180,E1 17998.081,E2 17998.081} C_VEL
LIN {X 0,Y 225.783,Z 678.81,A -85,B 0,C 180,E1 18013.603,E2 18013.603} C_VEL
LIN {X 0,Y 225.123,Z 678.81,A -85,B 0,C 180,E1 18019.558,E2 18019.558} C_VEL
LIN {X 0,Y 216.412,Z 678.81,A -85,B 0,C 180,E1 18028.505,E2 18028.505} C_VEL
LIN {X 0,Y 215.803,Z 678.81,A -85,B 0,C 180,E1 18042.408,E2 18042.408} C_VEL
LIN {X 0,Y 216.153,Z 678.81,A -85,B 0,C 180,E1 18058.227,E2 18058.227} C_VEL
LIN {X 0,Y 217.064,Z 680.051,A -85,B 0,C 180,E1 18070.286,E2 18070.286} C_VEL
LIN {X 0,Y 234.778,Z 721.02,A -85,B 0,C 180,E1 18076.472,E2 18076.472} C_VEL
LIN {X 0,Y 239.599,Z 755.125,A -85,B 0,C 180,E1 18082.265,E2 18082.265} C_VEL
LIN {X 0,Y 230.456,Z 790.442,A -85,B 0,C 180,E1 18090.472,E2 18090.472} C_VEL
LIN {X 0,Y 224.236,Z 812.516,A -85,B 0,C 180,E1 18101.101,E2 18101.101} C_VEL
LIN {X 0,Y 223.4,Z 820.791,A -85,B 0,C 180,E1 18113.504,E2 18113.504} C_VEL
LIN {X 0,Y 229.59,Z 814.429,A -85,B 0,C 180,E1 18125.335,E2 18125.335} C_VEL
LIN {X 0,Y 241.904,Z 793.815,A -85,B 0,C 180,E1 18135.567,E2 18135.567} C_VEL
LIN {X 0,Y 253.033,Z 766.77,A -85,B 0,C 180,E1 18142.255,E2 18142.255} C_VEL
LIN {X 0,Y 248.482,Z 734.796,A -85,B 0,C 180,E1 18150.655,E2 18150.655} C_VEL
LIN {X 0,Y 235.181,Z 705.445,A -85,B 0,C 180,E1 18160.383,E2 18160.383} C_VEL
LIN {X 0,Y 222.74,Z 686.095,A -85,B 0,C 180,E1 18170.691,E2 18170.691} C_VEL
LIN {X 0,Y 219.05,Z 678.81,A -85,B 0,C 180,E1 18178.019,E2 18178.019} C_VEL
LIN {X 0,Y 218.109,Z 680.672,A -85,B 0,C 180,E1 18192.323,E2 18192.323} C_VEL
LIN {X 0,Y 224.272,Z 690,A -85,B 0,C 180,E1 18200.828,E2 18200.828} C_VEL
LIN {X 0,Y 238.296,Z 709.611,A -85,B 0,C 180,E1 18210.729,E2 18210.729} C_VEL
LIN {X 0,Y 255.628,Z 743.019,A -85,B 0,C 180,E1 18219.795,E2 18219.795} C_VEL
LIN {X 0,Y 262.114,Z 770.737,A -85,B 0,C 180,E1 18224.87,E2 18224.87} C_VEL
LIN {X 0,Y 246.662,Z 815.751,A -85,B 0,C 180,E1 18230.62,E2 18230.62} C_VEL
LIN {X 0,Y 230.93,Z 851.774,A -85,B 0,C 180,E1 18239.956,E2 18239.956} C_VEL
LIN {X 0,Y 222.036,Z 875.266,A -85,B 0,C 180,E1 18252.088,E2 18252.088} C_VEL
LIN {X 0,Y 221.476,Z 885.032,A -85,B 0,C 180,E1 18264.101,E2 18264.101} C_VEL
LIN {X 0,Y 221.87,Z 883.953,A -85,B 0,C 180,E1 18273.922,E2 18273.922} C_VEL
LIN {X 0,Y 222.11,Z 868.976,A -85,B 0,C 180,E1 18286.735,E2 18286.735} C_VEL
LIN {X 0,Y 228.614,Z 839.613,A -85,B 0,C 180,E1 18298.226,E2 18298.226} C_VEL
LIN {X 0,Y 239.59,Z 798.301,A -85,B 0,C 180,E1 18306.71,E2 18306.71} C_VEL
LIN {X 0,Y 246.469,Z 758.4,A -85,B 0,C 180,E1 18311.177,E2 18311.177} C_VEL
LIN {X 0,Y 230.804,Z 709.76,A -85,B 0,C 180,E1 18316.656,E2 18316.656} C_VEL
LIN {X 0,Y 216.085,Z 678.81,A -85,B 0,C 180,E1 18321.009,E2 18321.009} C_VEL
LIN {X 0,Y 216.38,Z 678.81,A -85,B 0,C 180,E1 18332.873,E2 18332.873} C_VEL
LIN {X 0,Y 217.463,Z 678.81,A -85,B 0,C 180,E1 18345.858,E2 18345.858} C_VEL
LIN {X 0,Y 219.001,Z 678.81,A -85,B 0,C 180,E1 18358.01,E2 18358.01} C_VEL
LIN {X 0,Y 217.673,Z 678.81,A -85,B 0,C 180,E1 18374.12,E2 18374.12} C_VEL
LIN {X 0,Y 216.412,Z 678.81,A -85,B 0,C 180,E1 18388.505,E2 18388.505} C_VEL
LIN {X 0,Y 207.707,Z 678.81,A -85,B 0,C 180,E1 18397.847,E2 18397.847} C_VEL
LIN {X 0,Y 207.713,Z 678.81,A -85,B 0,C 180,E1 18411.61,E2 18411.61} C_VEL
LIN {X 0,Y 208.701,Z 678.81,A -85,B 0,C 180,E1 18428.146,E2 18428.146} C_VEL
LIN {X 0,Y 227.844,Z 723.404,A -85,B 0,C 180,E1 18435.584,E2 18435.584} C_VEL
LIN {X 0,Y 232.332,Z 756.722,A -85,B 0,C 180,E1 18441.552,E2 18441.552} C_VEL
LIN {X 0,Y 222.774,Z 791.758,A -85,B 0,C 180,E1 18450,E2 18450} C_VEL
LIN {X 0,Y 216.634,Z 812.497,A -85,B 0,C 180,E1 18460.086,E2 18460.086} C_VEL
LIN {X 0,Y 215.335,Z 821.856,A -85,B 0,C 180,E1 18472.806,E2 18472.806} C_VEL
LIN {X 0,Y 221.777,Z 816.213,A -85,B 0,C 180,E1 18485.565,E2 18485.565} C_VEL
LIN {X 0,Y 234.411,Z 796.611,A -85,B 0,C 180,E1 18496.073,E2 18496.073} C_VEL
LIN {X 0,Y 246.628,Z 768.98,A -85,B 0,C 180,E1 18503.31,E2 18503.31} C_VEL
LIN {X 0,Y 242.765,Z 737.837,A -85,B 0,C 180,E1 18512.044,E2 18512.044} C_VEL
